C05405=1042.762,309.484,-115.253,172.109,41.467,157.953
C05406=1042.769,309.732,-115.287,172.114,41.469,157.954
C05407=1042.775,309.979,-115.320,172.118,41.472,157.955
C05408=1042.783,310.227,-115.354,172.122,41.474,157.956
C05409=1042.790,310.474,-115.386,172.126,41.477,157.956
C05410=1042.798,310.722,-115.420,172.129,41.479,157.957
C05411=1042.804,310.969,-115.454,172.133,41.482,157.958
C05412=1042.811,311.217,-115.487,172.137,41.484,157.959
C05413=1042.819,311.464,-115.521,172.141,41.487,157.960
C05414=1042.825,311.713,-115.554,172.145,41.489,157.960
C05415=1042.833,311.960,-115.588,172.149,41.492,157.961
C05416=1042.839,312.207,-115.622,172.153,41.494,157.962
C05417=1042.846,312.455,-115.656,172.158,41.497,157.963
C05418=1042.854,312.703,-115.689,172.162,41.499,157.964
C05419=1042.860,312.951,-115.724,172.166,41.503,157.965
C05420=1042.867,313.198,-115.757,172.170,41.505,157.965
C05421=1042.873,313.446,-115.792,172.174,41.508,157.966
C05422=1042.880,313.693,-115.825,172.178,41.510,157.967
C05423=1042.886,313.940,-115.860,172.181,41.513,157.968
C05424=1042.894,314.188,-115.894,172.186,41.516,157.969
C05425=1042.900,314.436,-115.928,172.190,41.519,157.970
C05426=1042.907,314.683,-115.962,172.193,41.521,157.970
C05427=1042.915,314.931,-115.996,172.197,41.524,157.971
C05428=1042.921,315.178,-116.031,172.202,41.527,157.972
C05429=1042.928,315.425,-116.065,172.205,41.530,157.973
C05430=1042.934,315.673,-116.099,172.210,41.532,157.974
C05431=1042.942,315.921,-116.133,172.214,41.535,157.975
C05432=1042.948,316.168,-116.168,172.218,41.538,157.976
C05433=1042.955,316.415,-116.202,172.222,41.540,157.976
C05434=1042.961,316.663,-116.236,172.226,41.543,157.977
C05435=1042.969,316.911,-116.270,172.230,41.546,157.978
C05436=1042.975,317.158,-116.305,172.234,41.549,157.979
C05437=1042.983,317.406,-116.339,172.238,41.551,157.980
C05438=1042.989,317.653,-116.374,172.243,41.554,157.981
C05439=1042.997,317.901,-116.408,172.247,41.557,157.982
C05440=1043.003,318.149,-116.442,172.251,41.560,157.982
C05441=1043.011,318.396,-116.477,172.255,41.563,157.983
C05442=1043.016,318.643,-116.511,172.259,41.565,157.984
C05443=1043.024,318.890,-116.545,172.263,41.568,157.985
C05444=1043.033,319.226,-116.592,172.270,41.572,157.986
C05445=1043.042,319.561,-116.639,172.275,41.576,157.988
C05446=1043.052,319.896,-116.685,172.280,41.579,157.989
C05447=1043.062,320.232,-116.733,172.287,41.583,157.990
C05448=1043.069,320.479,-116.766,172.291,41.586,157.991
C05449=1043.076,320.727,-116.802,172.295,41.589,157.992
C05450=1043.082,320.975,-116.836,172.299,41.592,157.993
C05451=1043.090,321.222,-116.871,172.304,41.595,157.994
C05452=1043.096,321.469,-116.906,172.308,41.597,157.994
C05453=1043.104,321.717,-116.939,172.312,41.600,157.995
C05454=1043.110,321.964,-116.975,172.316,41.603,157.996
C05455=1043.118,322.211,-117.009,172.321,41.606,157.997
C05456=1043.124,322.459,-117.044,172.325,41.608,157.998
C05457=1043.132,322.706,-117.078,172.329,41.612,157.999
C05458=1043.139,322.954,-117.114,172.333,41.614,158.000
C05459=1043.146,323.202,-117.147,172.338,41.617,158.001
C05460=1043.153,323.449,-117.183,172.342,41.620,158.002
C05461=1043.160,323.697,-117.218,172.346,41.623,158.003
C05462=1043.167,323.944,-117.252,172.350,41.626,158.003
C05463=1043.174,324.192,-117.287,172.355,41.629,158.004
C05464=1043.181,324.439,-117.321,172.359,41.631,158.005
C05465=1043.189,324.687,-117.357,172.364,41.634,158.006
C05466=1043.196,324.934,-117.391,172.369,41.637,158.007
C05467=1043.203,325.181,-117.426,172.373,41.640,158.008
C05468=1043.210,325.429,-117.462,172.377,41.643,158.009
C05469=1043.218,325.677,-117.496,172.382,41.645,158.010
C05470=1043.225,325.924,-117.532,172.386,41.649,158.011
C05471=1043.232,326.171,-117.566,172.390,41.652,158.012
C05472=1043.239,326.419,-117.601,172.395,41.654,158.013
C05473=1043.247,326.667,-117.635,172.399,41.657,158.014
C05474=1043.254,326.914,-117.671,172.403,41.660,158.014
C05475=1043.260,327.161,-117.706,172.408,41.663,158.015
C05476=1043.268,327.408,-117.740,172.412,41.666,158.016
C05477=1043.275,327.656,-117.776,172.416,41.669,158.017
C05478=1043.283,327.903,-117.811,172.422,41.672,158.018
C05479=1043.290,328.150,-117.846,172.425,41.675,158.019
C05480=1043.297,328.398,-117.882,172.431,41.678,158.020
C05481=1043.305,328.645,-117.916,172.435,41.681,158.021
C05482=1043.312,328.894,-117.952,172.439,41.683,158.022
C05483=1043.319,329.141,-117.987,172.444,41.686,158.023
C05484=1043.326,329.388,-118.022,172.448,41.689,158.024
C05485=1043.334,329.635,-118.058,172.452,41.693,158.025
C05486=1043.341,329.883,-118.093,172.457,41.696,158.026
C05487=1043.348,330.130,-118.128,172.461,41.699,158.027
C05488=1043.355,330.378,-118.164,172.467,41.702,158.028
C05489=1043.362,330.625,-118.199,172.471,41.705,158.029
C05490=1043.369,330.872,-118.234,172.475,41.708,158.030
C05491=1043.376,331.120,-118.271,172.480,41.711,158.031
C05492=1043.382,331.367,-118.306,172.484,41.714,158.032
C05493=1043.389,331.614,-118.342,172.489,41.717,158.033
C05494=1043.397,331.862,-118.378,172.493,41.720,158.034
C05495=1043.404,332.109,-118.413,172.498,41.723,158.035
C05496=1043.411,332.357,-118.449,172.503,41.726,158.036
C05497=1043.418,332.604,-118.485,172.507,41.730,158.037
C05498=1043.425,332.851,-118.520,172.512,41.733,158.038
C05499=1043.433,333.099,-118.556,172.516,41.736,158.039
C05500=1043.443,333.428,-118.604,172.523,41.740,158.040
C05501=1043.452,333.760,-118.651,172.528,41.744,158.041
C05502=1043.462,334.090,-118.699,172.535,41.749,158.043
C05503=1043.472,334.420,-118.747,172.541,41.753,158.044
C05504=1043.479,334.667,-118.783,172.546,41.756,158.045
C05505=1043.486,334.915,-118.818,172.551,41.759,158.046
C05506=1043.493,335.162,-118.854,172.555,41.762,158.047
C05507=1043.501,335.409,-118.890,172.560,41.765,158.048
C05508=1043.508,335.656,-118.926,172.564,41.768,158.049
C05509=1043.515,335.904,-118.962,172.569,41.772,158.050
C05510=1043.522,336.151,-118.998,172.574,41.775,158.051
C05511=1043.529,336.399,-119.034,172.578,41.778,158.052
C05512=1043.536,336.645,-119.070,172.583,41.782,158.053
C05513=1043.543,336.893,-119.107,172.588,41.785,158.054
C05514=1043.550,337.140,-119.143,172.593,41.788,158.055
C05515=1043.558,337.387,-119.179,172.598,41.792,158.057
C05516=1043.565,337.635,-119.216,172.602,41.795,158.058
C05517=1043.572,337.882,-119.252,172.608,41.798,158.059
C05518=1043.580,338.129,-119.288,172.612,41.801,158.060
C05519=1043.588,338.377,-119.324,172.617,41.804,158.061
C05520=1043.594,338.624,-119.361,172.621,41.808,158.062
C05521=1043.602,338.871,-119.397,172.626,41.811,158.063
C05522=1043.609,339.118,-119.433,172.631,41.815,158.064
C05523=1043.616,339.366,-119.469,172.636,41.818,158.065
C05524=1043.623,339.613,-119.506,172.640,41.821,158.066
C05525=1043.631,339.861,-119.542,172.645,41.824,158.067
C05526=1043.637,340.108,-119.578,172.651,41.828,158.068
C05527=1043.645,340.355,-119.615,172.655,41.831,158.069
C05528=1043.653,340.602,-119.651,172.660,41.835,158.070
C05529=1043.660,340.849,-119.687,172.665,41.838,158.072
C05530=1043.667,341.096,-119.724,172.670,41.841,158.073
C05531=1043.675,341.344,-119.760,172.675,41.845,158.074
C05532=1043.682,341.591,-119.797,172.679,41.848,158.075
C05533=1043.689,341.838,-119.834,172.685,41.851,158.076
C05534=1043.697,342.085,-119.870,172.689,41.855,158.077
C05535=1043.704,342.333,-119.907,172.694,41.858,158.078
C05536=1043.711,342.580,-119.944,172.699,41.862,158.079
C05537=1043.718,342.828,-119.980,172.704,41.865,158.080
C05538=1043.726,343.074,-120.017,172.709,41.869,158.081
C05539=1043.733,343.321,-120.054,172.714,41.872,158.082
C05540=1043.741,343.568,-120.091,172.719,41.875,158.084
C05541=1043.748,343.816,-120.128,172.724,41.879,158.085
C05542=1043.755,344.063,-120.165,172.729,41.883,158.086
C05543=1043.762,344.310,-120.201,172.734,41.886,158.087
C05544=1043.769,344.557,-120.239,172.739,41.889,158.088
C05545=1043.777,344.804,-120.275,172.744,41.893,158.089
C05546=1043.784,345.052,-120.312,172.749,41.896,158.090
C05547=1043.792,345.299,-120.348,172.754,41.900,158.092
C05548=1043.799,345.546,-120.386,172.759,41.904,158.093
C05549=1043.806,345.793,-120.424,172.764,41.907,158.094
C05550=1043.814,346.041,-120.460,172.769,41.911,158.095
C05551=1043.821,346.288,-120.497,172.775,41.914,158.096
C05552=1043.828,346.534,-120.534,172.779,41.918,158.097
C05553=1043.836,346.781,-120.571,172.784,41.921,158.099
C05554=1043.843,347.029,-120.608,172.790,41.925,158.100
C05555=1043.850,347.276,-120.646,172.795,41.929,158.101
C05556=1043.860,347.603,-120.695,172.802,41.933,158.102
C05557=1043.870,347.929,-120.744,172.809,41.938,158.104
C05558=1043.880,348.256,-120.793,172.815,41.943,158.106
C05559=1043.890,348.583,-120.842,172.821,41.947,158.107
C05560=1043.897,348.830,-120.880,172.827,41.952,158.108
C05561=1043.905,349.077,-120.917,172.832,41.955,158.109
C05562=1043.912,349.324,-120.954,172.838,41.959,158.111
C05563=1043.920,349.571,-120.992,172.843,41.962,158.112
C05564=1043.927,349.818,-121.029,172.847,41.966,158.113
C05565=1043.935,350.065,-121.066,172.853,41.969,158.114
C05566=1043.942,350.312,-121.104,172.858,41.973,158.115
C05567=1043.949,350.559,-121.141,172.864,41.977,158.117
C05568=1043.957,350.807,-121.179,172.869,41.980,158.118
C05569=1043.965,351.054,-121.217,172.874,41.985,158.119
C05570=1043.972,351.301,-121.255,172.879,41.988,158.120
C05571=1043.979,351.548,-121.292,172.884,41.992,158.121
C05572=1043.987,351.795,-121.329,172.890,41.996,158.123
C05573=1043.994,352.042,-121.367,172.895,41.999,158.124
C05574=1044.002,352.288,-121.405,172.901,42.003,158.125
C05575=1044.009,352.535,-121.443,172.905,42.007,158.126
C05576=1044.017,352.783,-121.481,172.911,42.011,158.128
C05577=1044.025,353.030,-121.519,172.916,42.015,158.129
C05578=1044.032,353.277,-121.556,172.922,42.019,158.130
C05579=1044.039,353.523,-121.595,172.927,42.022,158.131
C05580=1044.047,353.771,-121.632,172.933,42.026,158.133
C05581=1044.055,354.018,-121.670,172.938,42.030,158.134
C05582=1044.062,354.265,-121.708,172.944,42.034,158.135
C05583=1044.069,354.512,-121.746,172.948,42.038,158.136
C05584=1044.077,354.759,-121.784,172.954,42.042,158.138
C05585=1044.085,355.006,-121.822,172.959,42.046,158.139
C05586=1044.092,355.253,-121.860,172.965,42.049,158.140
C05587=1044.100,355.500,-121.898,172.970,42.053,158.142
C05588=1044.107,355.747,-121.936,172.976,42.057,158.143
C05589=1044.115,355.994,-121.975,172.981,42.061,158.144
C05590=1044.122,356.241,-122.012,172.987,42.065,158.145
C05591=1044.131,356.487,-122.050,172.992,42.069,158.147
C05592=1044.139,356.734,-122.088,172.998,42.073,158.148
C05593=1044.145,356.982,-122.126,173.003,42.077,158.149
C05594=1044.153,357.228,-122.165,173.009,42.081,158.151
C05595=1044.161,357.475,-122.203,173.015,42.085,158.152
C05596=1044.169,357.722,-122.242,173.020,42.089,158.153
C05597=1044.177,357.970,-122.279,173.026,42.093,158.155
C05598=1044.184,358.216,-122.318,173.031,42.096,158.156
C05599=1044.192,358.463,-122.356,173.037,42.100,158.157
C05600=1044.199,358.710,-122.395,173.042,42.105,158.158
C05601=1044.207,358.957,-122.433,173.048,42.109,158.160
C05602=1044.215,359.204,-122.472,173.054,42.113,158.161
C05603=1044.222,359.451,-122.510,173.059,42.117,158.162
C05604=1044.230,359.698,-122.549,173.065,42.121,158.164
C05605=1044.238,359.944,-122.587,173.070,42.125,158.165
C05606=1044.245,360.191,-122.626,173.076,42.129,158.166
C05607=1044.253,360.438,-122.665,173.082,42.133,158.168
C05608=1044.261,360.685,-122.703,173.087,42.138,158.169
C05609=1044.269,360.932,-122.741,173.093,42.142,158.171
C05610=1044.276,361.180,-122.781,173.099,42.146,158.172
C05611=1044.284,361.426,-122.820,173.104,42.150,158.173
C05612=1044.294,361.758,-122.871,173.112,42.155,158.175
C05613=1044.305,362.091,-122.923,173.120,42.161,158.177
C05614=1044.315,362.423,-122.976,173.128,42.166,158.179
C05615=1044.326,362.755,-123.028,173.135,42.172,158.181
C05616=1044.333,363.003,-123.068,173.141,42.177,158.182
C05617=1044.341,363.249,-123.106,173.147,42.181,158.184
C05618=1044.349,363.496,-123.146,173.153,42.185,158.185
C05619=1044.356,363.743,-123.184,173.159,42.189,158.186
C05620=1044.365,363.989,-123.223,173.165,42.193,158.188
C05621=1044.372,364.237,-123.262,173.170,42.198,158.189
C05622=1044.380,364.483,-123.301,173.176,42.202,158.191
C05623=1044.387,364.730,-123.341,173.182,42.206,158.192
C05624=1044.396,364.977,-123.380,173.187,42.211,158.193
C05625=1044.403,365.223,-123.420,173.194,42.215,158.195
C05626=1044.411,365.470,-123.458,173.200,42.219,158.196
C05627=1044.419,365.717,-123.498,173.206,42.224,158.198
C05628=1044.425,365.964,-123.537,173.212,42.228,158.199
C05629=1044.434,366.210,-123.576,173.217,42.232,158.201
C05630=1044.442,366.457,-123.616,173.223,42.237,158.202
C05631=1044.450,366.703,-123.655,173.230,42.241,158.204
C05632=1044.457,366.951,-123.694,173.235,42.245,158.205
C05633=1044.465,367.197,-123.734,173.241,42.250,158.207
C05634=1044.473,367.444,-123.774,173.247,42.255,158.208
C05635=1044.482,367.691,-123.813,173.254,42.258,158.209
C05636=1044.489,367.937,-123.852,173.260,42.263,158.211
C05637=1044.497,368.184,-123.892,173.265,42.268,158.212
C05638=1044.505,368.431,-123.931,173.271,42.272,158.214
C05639=1044.513,368.678,-123.970,173.278,42.277,158.215
C05640=1044.521,368.925,-124.010,173.284,42.281,158.217
C05641=1044.529,369.171,-124.050,173.289,42.285,158.218
C05642=1044.537,369.418,-124.089,173.296,42.290,158.220
C05643=1044.545,369.665,-124.129,173.302,42.294,158.221
C05644=1044.552,369.911,-124.168,173.308,42.299,158.223
C05645=1044.560,370.158,-124.208,173.314,42.303,158.224
C05646=1044.569,370.404,-124.248,173.321,42.308,158.226
C05647=1044.577,370.651,-124.288,173.327,42.312,158.227
C05648=1044.585,370.897,-124.328,173.333,42.317,158.229
C05649=1044.593,371.144,-124.367,173.339,42.321,158.230
C05650=1044.601,371.391,-124.407,173.345,42.327,158.232
C05651=1044.609,371.637,-124.448,173.352,42.331,158.234
C05652=1044.616,371.884,-124.488,173.358,42.336,158.235
C05653=1044.624,372.131,-124.528,173.364,42.340,158.237
C05654=1044.633,372.377,-124.568,173.371,42.345,158.238
C05655=1044.641,372.624,-124.608,173.377,42.350,158.240
C05656=1044.649,372.870,-124.648,173.383,42.354,158.241
C05657=1044.656,373.117,-124.688,173.389,42.359,158.243
C05658=1044.664,373.364,-124.729,173.395,42.364,158.245
C05659=1044.672,373.611,-124.769,173.402,42.368,158.246
C05660=1044.680,373.857,-124.810,173.408,42.373,158.248
C05661=1044.688,374.104,-124.849,173.414,42.378,158.249
C05662=1044.697,374.350,-124.889,173.421,42.383,158.251
C05663=1044.705,374.597,-124.930,173.427,42.388,158.253
C05664=1044.713,374.844,-124.970,173.434,42.393,158.254
C05665=1044.721,375.090,-125.011,173.440,42.397,158.256
C05666=1044.729,375.336,-125.052,173.447,42.402,158.258
C05667=1044.737,375.583,-125.092,173.453,42.407,158.259
C05668=1044.748,375.935,-125.150,173.462,42.414,158.261
C05669=1044.760,376.287,-125.207,173.472,42.421,158.264
C05670=1044.772,376.639,-125.266,173.481,42.427,158.266
C05671=1044.783,376.991,-125.324,173.490,42.434,158.268
C05672=1044.792,377.237,-125.364,173.497,42.439,158.270
C05673=1044.800,377.483,-125.404,173.504,42.444,158.272
C05674=1044.809,377.730,-125.445,173.510,42.449,158.273
C05675=1044.817,377.976,-125.486,173.517,42.454,158.275
C05676=1044.825,378.223,-125.527,173.524,42.459,158.277
C05677=1044.833,378.470,-125.568,173.530,42.464,158.278
C05678=1044.841,378.716,-125.608,173.537,42.469,158.280
C05679=1044.849,378.962,-125.649,173.543,42.474,158.282
C05680=1044.858,379.209,-125.690,173.550,42.479,158.283
C05681=1044.866,379.455,-125.730,173.557,42.484,158.285
C05682=1044.874,379.702,-125.771,173.563,42.489,158.287
C05683=1044.882,379.948,-125.813,173.570,42.494,158.289
C05684=1044.890,380.195,-125.854,173.576,42.499,158.290
C05685=1044.898,380.441,-125.895,173.584,42.504,158.292
C05686=1044.907,380.687,-125.936,173.591,42.509,158.294
C05687=1044.915,380.934,-125.978,173.597,42.514,158.296
C05688=1044.924,381.180,-126.019,173.604,42.519,158.297
C05689=1044.932,381.427,-126.060,173.610,42.525,158.299
C05690=1044.940,381.674,-126.101,173.617,42.530,158.301
C05691=1044.948,381.920,-126.143,173.624,42.535,158.303
C05692=1044.956,382.165,-126.184,173.632,42.540,158.304
C05693=1044.965,382.412,-126.225,173.638,42.545,158.306
C05694=1044.973,382.658,-126.267,173.645,42.550,158.308
C05695=1044.981,382.905,-126.308,173.652,42.556,158.310
C05696=1044.990,383.151,-126.350,173.658,42.561,158.311
C05697=1044.998,383.397,-126.391,173.666,42.566,158.313
C05698=1045.006,383.644,-126.433,173.673,42.571,158.315
C05699=1045.014,383.890,-126.474,173.680,42.577,158.317
C05700=1045.023,384.136,-126.516,173.686,42.582,158.319
C05701=1045.032,384.382,-126.557,173.694,42.587,158.320
C05702=1045.040,384.629,-126.599,173.701,42.593,158.322
C05703=1045.049,384.876,-126.641,173.708,42.598,158.324
C05704=1045.057,385.121,-126.682,173.714,42.603,158.326
C05705=1045.065,385.368,-126.724,173.722,42.609,158.328
C05706=1045.074,385.615,-126.766,173.729,42.614,158.330
C05707=1045.082,385.860,-126.807,173.736,42.620,158.332
C05708=1045.091,386.107,-126.849,173.743,42.625,158.333
C05709=1045.099,386.353,-126.891,173.751,42.630,158.335
C05710=1045.108,386.600,-126.933,173.757,42.636,158.337
C05711=1045.117,386.845,-126.974,173.764,42.641,158.339
C05712=1045.125,387.092,-127.017,173.772,42.647,158.341
C05713=1045.134,387.338,-127.058,173.779,42.652,158.343
C05714=1045.143,387.585,-127.100,173.786,42.658,158.345
C05715=1045.151,387.831,-127.143,173.794,42.663,158.347
C05716=1045.160,388.077,-127.185,173.801,42.669,158.348
C05717=1045.169,388.323,-127.226,173.808,42.674,158.350
C05718=1045.177,388.569,-127.269,173.816,42.679,158.352
C05719=1045.186,388.815,-127.311,173.823,42.685,158.354
C05720=1045.194,389.062,-127.353,173.831,42.691,158.356
C05721=1045.203,389.308,-127.395,173.838,42.696,158.358
C05722=1045.212,389.554,-127.438,173.844,42.702,158.360
C05723=1045.220,389.801,-127.480,173.852,42.708,158.362
C05724=1045.231,390.093,-127.531,173.861,42.714,158.364
C05725=1045.241,390.386,-127.581,173.870,42.721,158.367
C05726=1045.251,390.679,-127.632,173.879,42.728,158.369
C05727=1045.261,390.971,-127.682,173.888,42.735,158.371
C05728=1045.270,391.218,-127.725,173.895,42.740,158.373
C05729=1045.279,391.464,-127.767,173.903,42.746,158.375
C05730=1045.287,391.710,-127.810,173.910,42.752,158.377
C05731=1045.296,391.956,-127.853,173.917,42.758,158.379
C05732=1045.305,392.202,-127.895,173.925,42.763,158.381
C05733=1045.313,392.448,-127.938,173.934,42.769,158.383
C05734=1045.322,392.694,-127.981,173.941,42.775,158.385
C05735=1045.331,392.941,-128.024,173.949,42.781,158.387
C05736=1045.340,393.187,-128.067,173.956,42.787,158.389
C05737=1045.349,393.433,-128.110,173.964,42.793,158.391
C05738=1045.357,393.679,-128.153,173.971,42.799,158.394
C05739=1045.366,393.925,-128.196,173.979,42.805,158.396
C05740=1045.375,394.171,-128.238,173.987,42.811,158.398
C05741=1045.383,394.417,-128.281,173.994,42.817,158.400
C05742=1045.392,394.663,-128.325,174.003,42.822,158.402
C05743=1045.401,394.910,-128.368,174.010,42.828,158.404
C05744=1045.411,395.155,-128.411,174.018,42.834,158.406
C05745=1045.419,395.401,-128.454,174.026,42.840,158.408
C05746=1045.428,395.647,-128.497,174.033,42.846,158.410
C05747=1045.437,395.893,-128.540,174.042,42.852,158.412
C05748=1045.445,396.139,-128.584,174.050,42.858,158.414
C05749=1045.454,396.385,-128.627,174.057,42.864,158.417
C05750=1045.463,396.631,-128.671,174.065,42.871,158.419
C05751=1045.472,396.877,-128.714,174.074,42.877,158.421
C05752=1045.481,397.123,-128.758,174.081,42.883,158.423
C05753=1045.490,397.369,-128.801,174.089,42.889,158.425
C05754=1045.499,397.615,-128.845,174.097,42.895,158.427
C05755=1045.508,397.862,-128.889,174.106,42.901,158.430
C05756=1045.516,398.107,-128.932,174.114,42.908,158.432
C05757=1045.526,398.352,-128.975,174.121,42.914,158.434
C05758=1045.535,398.599,-129.019,174.130,42.920,158.436
C05759=1045.544,398.844,-129.063,174.138,42.926,158.438
C05760=1045.553,399.090,-129.107,174.145,42.932,158.440
C05761=1045.562,399.336,-129.150,174.154,42.939,158.443
C05762=1045.571,399.583,-129.194,174.162,42.945,158.445
C05763=1045.580,399.828,-129.238,174.171,42.952,158.447
C05764=1045.589,400.074,-129.282,174.179,42.957,158.449
C05765=1045.599,400.320,-129.326,174.187,42.964,158.452
C05766=1045.608,400.566,-129.370,174.195,42.970,158.454
C05767=1045.616,400.812,-129.414,174.203,42.977,158.456
C05768=1045.625,401.058,-129.458,174.212,42.983,158.458
C05769=1045.635,401.304,-129.502,174.220,42.989,158.461
C05770=1045.644,401.550,-129.546,174.229,42.996,158.463
C05771=1045.653,401.795,-129.590,174.237,43.003,158.465
C05772=1045.662,402.041,-129.634,174.246,43.009,158.468
C05773=1045.671,402.287,-129.679,174.254,43.015,158.470
C05774=1045.681,402.533,-129.724,174.263,43.022,158.472
C05775=1045.689,402.779,-129.767,174.271,43.029,158.475
C05776=1045.702,403.117,-129.829,174.283,43.037,158.478
C05777=1045.715,403.456,-129.890,174.294,43.047,158.481
C05778=1045.728,403.793,-129.951,174.306,43.056,158.484
C05779=1045.740,404.131,-130.012,174.318,43.065,158.488
C05780=1045.756,404.536,-130.086,174.332,43.076,158.492
C05781=1045.770,404.941,-130.160,174.346,43.087,158.496
C05782=1045.786,405.345,-130.233,174.360,43.098,158.500
C05783=1045.802,405.749,-130.307,174.376,43.109,158.504
C05784=1045.810,405.995,-130.353,174.384,43.116,158.506
C05785=1045.820,406.241,-130.397,174.393,43.123,158.508
C05786=1045.829,406.487,-130.442,174.402,43.130,158.511
C05787=1045.839,406.732,-130.487,174.410,43.137,158.513
C05788=1045.848,406.978,-130.532,174.419,43.144,158.516
C05789=1045.857,407.223,-130.577,174.428,43.150,158.518
C05790=1045.866,407.469,-130.623,174.438,43.157,158.521
C05791=1045.876,407.715,-130.667,174.447,43.164,158.523
C05792=1045.885,407.961,-130.713,174.455,43.172,158.526
C05793=1045.895,408.206,-130.758,174.464,43.178,158.528
C05794=1045.904,408.452,-130.802,174.473,43.185,158.531
C05795=1045.914,408.697,-130.849,174.483,43.192,158.533
C05796=1045.924,408.943,-130.894,174.492,43.199,158.536
C05797=1045.933,409.189,-130.939,174.500,43.207,158.539
C05798=1045.943,409.434,-130.984,174.509,43.213,158.541
C05799=1045.952,409.680,-131.030,174.519,43.221,158.544
C05800=1045.962,409.926,-131.075,174.528,43.228,158.546
C05801=1045.971,410.172,-131.121,174.537,43.235,158.549
C05802=1045.981,410.417,-131.166,174.547,43.242,158.552
C05803=1045.991,410.663,-131.212,174.556,43.249,158.554
C05804=1046.001,410.908,-131.258,174.565,43.256,158.557
C05805=1046.010,411.155,-131.303,174.575,43.263,158.559
C05806=1046.020,411.400,-131.350,174.584,43.271,158.562
C05807=1046.030,411.645,-131.395,174.594,43.278,158.565
C05808=1046.039,411.891,-131.441,174.603,43.285,158.567
C05809=1046.050,412.137,-131.487,174.613,43.292,158.570
C05810=1046.059,412.383,-131.532,174.622,43.300,158.573
C05811=1046.070,412.628,-131.578,174.631,43.307,158.575
C05812=1046.079,412.873,-131.624,174.641,43.315,158.578
C05813=1046.089,413.119,-131.671,174.650,43.322,158.581
C05814=1046.098,413.364,-131.717,174.661,43.329,158.583
C05815=1046.108,413.610,-131.763,174.671,43.337,158.586
C05816=1046.117,413.856,-131.810,174.680,43.344,158.589
C05817=1046.128,414.101,-131.855,174.690,43.352,158.592
C05818=1046.137,414.346,-131.902,174.699,43.359,158.594
C05819=1046.147,414.592,-131.948,174.709,43.367,158.597
C05820=1046.157,414.838,-131.995,174.719,43.375,158.600
C05821=1046.166,415.083,-132.041,174.729,43.382,158.603
C05822=1046.176,415.329,-132.088,174.739,43.389,158.606
C05823=1046.186,415.575,-132.134,174.748,43.397,158.608
C05824=1046.197,415.819,-132.181,174.758,43.405,158.611
C05825=1046.206,416.065,-132.227,174.769,43.412,158.614
C05826=1046.217,416.310,-132.274,174.778,43.420,158.617
C05827=1046.227,416.556,-132.321,174.788,43.428,158.620
C05828=1046.236,416.801,-132.368,174.799,43.436,158.623
C05829=1046.246,417.046,-132.414,174.809,43.443,158.626
C05830=1046.256,417.292,-132.461,174.818,43.451,158.628
C05831=1046.266,417.538,-132.508,174.829,43.459,158.631
C05832=1046.277,417.783,-132.555,174.839,43.466,158.634
C05833=1046.287,418.028,-132.602,174.850,43.474,158.637
C05834=1046.297,418.274,-132.648,174.859,43.482,158.640
C05835=1046.307,418.519,-132.695,174.870,43.490,158.643
C05836=1046.324,418.930,-132.775,174.888,43.503,158.648
C05837=1046.341,419.343,-132.855,174.904,43.517,158.653
C05838=1046.358,419.754,-132.934,174.922,43.530,158.658
C05839=1046.375,420.166,-133.014,174.940,43.544,158.663
C05840=1046.386,420.412,-133.061,174.951,43.552,158.666
C05841=1046.396,420.657,-133.108,174.962,43.560,158.669
C05842=1046.405,420.902,-133.156,174.972,43.568,158.672
C05843=1046.416,421.147,-133.204,174.983,43.576,158.676
C05844=1046.426,421.392,-133.251,174.994,43.584,158.679
C05845=1046.436,421.638,-133.298,175.004,43.593,158.682
C05846=1046.447,421.883,-133.347,175.015,43.601,158.685
C05847=1046.457,422.128,-133.394,175.026,43.609,158.688
C05848=1046.467,422.373,-133.442,175.036,43.617,158.691
C05849=1046.477,422.619,-133.490,175.047,43.625,158.694
C05850=1046.489,422.864,-133.538,175.058,43.634,158.697
C05851=1046.499,423.109,-133.586,175.069,43.642,158.700
C05852=1046.509,423.354,-133.633,175.080,43.651,158.704
C05853=1046.520,423.599,-133.681,175.090,43.659,158.707
C05854=1046.530,423.844,-133.730,175.102,43.667,158.710
C05855=1046.541,424.090,-133.778,175.113,43.676,158.713
C05856=1046.552,424.334,-133.826,175.124,43.684,158.717
C05857=1046.562,424.580,-133.874,175.135,43.693,158.720
C05858=1046.572,424.825,-133.922,175.147,43.701,158.723
C05859=1046.583,425.071,-133.970,175.158,43.710,158.726
C05860=1046.594,425.315,-134.019,175.169,43.718,158.730
C05861=1046.604,425.560,-134.068,175.181,43.727,158.733
C05862=1046.615,425.805,-134.116,175.192,43.735,158.736
C05863=1046.625,426.051,-134.165,175.203,43.744,158.739
C05864=1046.636,426.296,-134.213,175.215,43.753,158.743
C05865=1046.647,426.540,-134.262,175.226,43.761,158.746
C05866=1046.658,426.786,-134.311,175.238,43.770,158.750
C05867=1046.668,427.030,-134.359,175.249,43.779,158.753
C05868=1046.679,427.275,-134.408,175.261,43.788,158.756
C05869=1046.690,427.520,-134.457,175.273,43.797,158.760
C05870=1046.701,427.766,-134.506,175.284,43.805,158.763
C05871=1046.711,428.010,-134.555,175.296,43.814,158.767
C05872=1046.723,428.255,-134.604,175.308,43.823,158.770
C05873=1046.733,428.500,-134.653,175.319,43.832,158.773
C05874=1046.744,428.745,-134.702,175.332,43.841,158.777
C05875=1046.755,428.990,-134.751,175.343,43.850,158.780
C05876=1046.766,429.235,-134.801,175.355,43.859,158.784
C05877=1046.777,429.479,-134.850,175.368,43.868,158.787
C05878=1046.787,429.724,-134.899,175.379,43.877,158.791
C05879=1046.798,429.969,-134.949,175.391,43.886,158.794
C05880=1046.809,430.214,-134.998,175.404,43.895,158.798
C05881=1046.820,430.459,-135.047,175.416,43.904,158.802
C05882=1046.831,430.704,-135.097,175.427,43.914,158.805
C05883=1046.842,430.948,-135.147,175.440,43.922,158.809
C05884=1046.853,431.193,-135.196,175.452,43.932,158.812
C05885=1046.864,431.438,-135.246,175.465,43.941,158.816
C05886=1046.875,431.683,-135.296,175.477,43.951,158.820
C05887=1046.886,431.928,-135.345,175.490,43.960,158.823
C05888=1046.897,432.172,-135.396,175.502,43.969,158.827
C05889=1046.908,432.418,-135.446,175.514,43.979,158.831
C05890=1046.920,432.662,-135.495,175.527,43.988,158.835
C05891=1046.931,432.907,-135.545,175.539,43.997,158.838
C05892=1046.941,433.124,-135.590,175.551,44.006,158.841
C05893=1046.951,433.342,-135.634,175.562,44.014,158.845
C05894=1046.961,433.559,-135.679,175.573,44.022,158.848
C05895=1046.971,433.776,-135.724,175.585,44.030,158.851
C05896=1046.981,433.993,-135.767,175.596,44.039,158.855
C05897=1046.991,434.210,-135.812,175.608,44.048,158.858
C05898=1047.001,434.428,-135.857,175.618,44.056,158.862
C05899=1047.012,434.644,-135.902,175.630,44.065,158.865
C05900=1047.023,434.889,-135.952,175.643,44.074,158.869
C05901=1047.034,435.134,-136.003,175.656,44.084,158.873
C05902=1047.045,435.378,-136.053,175.669,44.094,158.877
C05903=1047.058,435.623,-136.103,175.683,44.103,158.880
C05904=1047.069,435.868,-136.154,175.696,44.113,158.884
C05905=1047.080,436.112,-136.205,175.709,44.123,158.888
C05906=1047.092,436.357,-136.256,175.722,44.133,158.892
C05907=1047.103,436.601,-136.307,175.736,44.142,158.896
C05908=1047.115,436.846,-136.357,175.749,44.152,158.900
C05909=1047.126,437.090,-136.408,175.762,44.162,158.904
C05910=1047.138,437.335,-136.459,175.776,44.172,158.908
C05911=1047.150,437.580,-136.511,175.789,44.182,158.912
C05912=1047.161,437.824,-136.562,175.803,44.192,158.916
C05913=1047.173,438.068,-136.613,175.817,44.202,158.920
C05914=1047.184,438.313,-136.664,175.831,44.212,158.925
C05915=1047.196,438.558,-136.715,175.844,44.223,158.929
C05916=1047.208,438.802,-136.766,175.858,44.233,158.933
C05917=1047.219,439.046,-136.818,175.872,44.243,158.937
C05918=1047.232,439.290,-136.870,175.886,44.253,158.941
C05919=1047.243,439.534,-136.921,175.900,44.263,158.945
C05920=1047.255,439.779,-136.972,175.914,44.273,158.949
C05921=1047.267,440.023,-137.024,175.928,44.283,158.954
C05922=1047.279,440.268,-137.075,175.941,44.294,158.958
C05923=1047.291,440.512,-137.127,175.956,44.304,158.962
C05924=1047.303,440.756,-137.179,175.970,44.314,158.966
C05925=1047.315,441.000,-137.231,175.985,44.325,158.971
C05926=1047.327,441.245,-137.282,175.998,44.335,158.975
C05927=1047.339,441.490,-137.335,176.013,44.346,158.979
C05928=1047.351,441.733,-137.388,176.028,44.356,158.984
C05929=1047.363,441.978,-137.439,176.042,44.367,158.988
C05930=1047.376,442.222,-137.491,176.057,44.378,158.992
C05931=1047.388,442.466,-137.543,176.071,44.388,158.997
C05932=1047.399,442.710,-137.596,176.086,44.399,159.001
C05933=1047.412,442.955,-137.648,176.101,44.409,159.006
C05934=1047.424,443.198,-137.700,176.116,44.420,159.010
C05935=1047.436,443.442,-137.753,176.130,44.431,159.014
C05936=1047.448,443.687,-137.806,176.145,44.442,159.019
C05937=1047.461,443.931,-137.858,176.160,44.452,159.023
C05938=1047.473,444.174,-137.911,176.175,44.463,159.028
C05939=1047.486,444.419,-137.963,176.191,44.474,159.033
C05940=1047.497,444.663,-138.016,176.206,44.485,159.037
C05941=1047.510,444.907,-138.069,176.221,44.496,159.042
C05942=1047.523,445.151,-138.121,176.236,44.507,159.046
C05943=1047.536,445.395,-138.174,176.252,44.518,159.051
C05944=1047.548,445.638,-138.227,176.267,44.529,159.056
C05945=1047.561,445.880,-138.279,176.282,44.540,159.060
C05946=1047.575,446.124,-138.332,176.298,44.550,159.065
C05947=1047.589,446.368,-138.383,176.314,44.561,159.069
C05948=1047.604,446.612,-138.434,176.330,44.571,159.074
C05949=1047.620,446.855,-138.484,176.345,44.582,159.078
C05950=1047.636,447.099,-138.534,176.361,44.592,159.083
C05951=1047.654,447.343,-138.583,176.377,44.602,159.087
C05952=1047.680,447.713,-138.657,176.401,44.617,159.094
C05953=1047.709,448.082,-138.729,176.425,44.632,159.101
C05954=1047.739,448.452,-138.800,176.450,44.646,159.107
C05955=1047.771,448.823,-138.871,176.474,44.660,159.114
C05956=1047.793,449.067,-138.917,176.491,44.669,159.118
C05957=1047.815,449.312,-138.962,176.508,44.678,159.122
C05958=1047.838,449.558,-139.006,176.525,44.687,159.126
C05959=1047.862,449.802,-139.051,176.541,44.696,159.131
C05960=1047.886,450.048,-139.094,176.558,44.704,159.135
C05961=1047.911,450.294,-139.138,176.575,44.713,159.139
C05962=1047.937,450.539,-139.180,176.592,44.721,159.143
C05963=1047.964,450.783,-139.222,176.609,44.729,159.147
C05964=1047.654,450.817,-139.527,176.610,44.817,159.173
C05965=1047.628,450.571,-139.485,176.593,44.809,159.169
C05966=1047.602,450.325,-139.443,176.575,44.801,159.165
C05967=1047.576,450.080,-139.399,176.559,44.792,159.161
C05968=1047.552,449.835,-139.356,176.542,44.784,159.157
C05969=1047.528,449.590,-139.312,176.525,44.775,159.152
C05970=1047.505,449.344,-139.267,176.508,44.767,159.148
C05971=1047.482,449.100,-139.222,176.492,44.757,159.144
C05972=1047.460,448.854,-139.176,176.475,44.748,159.140
C05973=1047.430,448.502,-139.110,176.451,44.735,159.133
C05974=1047.401,448.149,-139.042,176.428,44.722,159.127
C05975=1047.373,447.797,-138.973,176.404,44.708,159.121
C05976=1047.346,447.445,-138.904,176.381,44.694,159.114
C05977=1047.330,447.201,-138.854,176.365,44.684,159.110
C05978=1047.312,446.957,-138.804,176.349,44.674,159.105
C05979=1047.296,446.713,-138.754,176.333,44.664,159.101
C05980=1047.280,446.469,-138.704,176.317,44.654,159.096
C05981=1047.266,446.226,-138.653,176.302,44.643,159.092
C05982=1047.252,445.982,-138.601,176.287,44.632,159.087
C05983=1047.239,445.739,-138.549,176.270,44.622,159.083
C05984=1047.225,445.496,-138.497,176.255,44.611,159.078
C05985=1047.213,445.252,-138.444,176.240,44.600,159.073
C05986=1047.201,445.008,-138.390,176.224,44.589,159.069
C05987=1047.188,444.764,-138.338,176.209,44.578,159.064
C05988=1047.175,444.520,-138.285,176.194,44.567,159.060
C05989=1047.163,444.276,-138.233,176.179,44.557,159.055
C05990=1047.150,444.032,-138.180,176.164,44.546,159.051
C05991=1047.139,443.788,-138.127,176.148,44.535,159.046
C05992=1047.126,443.544,-138.074,176.133,44.524,159.041
C05993=1047.114,443.300,-138.022,176.118,44.514,159.037
C05994=1047.101,443.056,-137.970,176.103,44.503,159.033
C05995=1047.089,442.811,-137.917,176.089,44.493,159.028
C05996=1047.077,442.567,-137.865,176.074,44.482,159.024
C05997=1047.065,442.323,-137.813,176.059,44.471,159.019
C05998=1047.053,442.079,-137.761,176.044,44.461,159.015
C05999=1047.041,441.835,-137.709,176.030,44.450,159.010
C06000=1047.028,441.590,-137.655,176.015,44.440,159.006
C06001=1047.017,441.346,-137.604,176.000,44.429,159.002
C06002=1047.004,441.102,-137.552,175.986,44.419,158.997
C06003=1046.993,440.858,-137.501,175.972,44.409,158.993
C06004=1046.980,440.614,-137.448,175.958,44.398,158.989
C06005=1046.968,440.369,-137.397,175.943,44.388,158.985
C06006=1046.956,440.125,-137.345,175.929,44.378,158.980
C06007=1046.944,439.881,-137.293,175.915,44.368,158.976
C06008=1046.933,439.636,-137.242,175.901,44.357,158.972
C06009=1046.920,439.392,-137.190,175.887,44.347,158.968
C06010=1046.908,439.148,-137.139,175.873,44.337,158.964
C06011=1046.897,438.903,-137.087,175.859,44.327,158.959
C06012=1046.885,438.659,-137.035,175.845,44.317,158.955
C06013=1046.874,438.414,-136.984,175.831,44.307,158.951
C06014=1046.862,438.170,-136.933,175.818,44.297,158.947
C06015=1046.850,437.926,-136.881,175.804,44.287,158.943
C06016=1046.839,437.681,-136.831,175.790,44.277,158.939
C06017=1046.826,437.436,-136.780,175.776,44.267,158.935
C06018=1046.815,437.193,-136.729,175.763,44.257,158.931
C06019=1046.803,436.948,-136.677,175.749,44.247,158.927
C06020=1046.791,436.703,-136.627,175.736,44.238,158.923
C06021=1046.780,436.459,-136.576,175.723,44.228,158.919
C06022=1046.769,436.214,-136.525,175.709,44.218,158.915
C06023=1046.757,435.970,-136.474,175.696,44.208,158.911
C06024=1046.746,435.725,-136.423,175.683,44.198,158.907
C06025=1046.734,435.480,-136.372,175.669,44.189,158.903
C06026=1046.722,435.236,-136.323,175.656,44.180,158.899
C06027=1046.711,434.991,-136.271,175.643,44.170,158.895
C06028=1046.700,434.747,-136.221,175.630,44.160,158.892
C06029=1046.689,434.528,-136.176,175.618,44.152,158.888
C06030=1046.679,434.311,-136.131,175.607,44.143,158.885
C06031=1046.669,434.092,-136.086,175.595,44.135,158.881
C06032=1046.658,433.874,-136.042,175.584,44.127,158.878
C06033=1046.649,433.656,-135.997,175.572,44.118,158.875
C06034=1046.638,433.438,-135.952,175.560,44.109,158.871
C06035=1046.628,433.219,-135.907,175.549,44.101,158.868
C06036=1046.618,433.001,-135.863,175.539,44.093,158.865
C06037=1046.607,432.757,-135.812,175.526,44.083,158.861
C06038=1046.595,432.512,-135.763,175.513,44.074,158.857
C06039=1046.585,432.267,-135.713,175.501,44.065,158.853
C06040=1046.574,432.022,-135.663,175.488,44.055,158.850
C06041=1046.562,431.777,-135.613,175.475,44.046,158.846
C06042=1046.551,431.532,-135.564,175.463,44.037,158.842
C06043=1046.540,431.288,-135.513,175.450,44.028,158.839
C06044=1046.529,431.043,-135.464,175.438,44.019,158.835
C06045=1046.518,430.798,-135.415,175.425,44.009,158.831
C06046=1046.507,430.554,-135.364,175.414,44.000,158.828
C06047=1046.496,430.309,-135.315,175.401,43.991,158.824
C06048=1046.485,430.064,-135.266,175.389,43.982,158.821
C06049=1046.474,429.819,-135.216,175.376,43.973,158.817
C06050=1046.463,429.574,-135.167,175.365,43.964,158.814
C06051=1046.452,429.329,-135.118,175.353,43.955,158.810
C06052=1046.442,429.085,-135.068,175.340,43.946,158.807
C06053=1046.431,428.840,-135.019,175.329,43.937,158.803
C06054=1046.420,428.595,-134.970,175.317,43.928,158.800
C06055=1046.409,428.350,-134.920,175.304,43.920,158.796
C06056=1046.398,428.105,-134.872,175.293,43.911,158.793
C06057=1046.387,427.860,-134.822,175.281,43.902,158.789
C06058=1046.376,427.615,-134.773,175.270,43.893,158.786
C06059=1046.366,427.370,-134.725,175.257,43.885,158.782
C06060=1046.355,427.125,-134.676,175.246,43.876,158.779
C06061=1046.344,426.880,-134.627,175.234,43.867,158.776
C06062=1046.333,426.635,-134.578,175.223,43.859,158.772
C06063=1046.323,426.390,-134.530,175.211,43.850,158.769
C06064=1046.312,426.144,-134.481,175.200,43.841,158.766
C06065=1046.301,425.900,-134.432,175.189,43.833,158.762
C06066=1046.290,425.655,-134.384,175.177,43.824,158.759
C06067=1046.280,425.409,-134.335,175.166,43.815,158.755
C06068=1046.270,425.165,-134.287,175.154,43.807,158.752
C06069=1046.259,424.920,-134.238,175.143,43.798,158.749
C06070=1046.248,424.675,-134.190,175.132,43.790,158.746
C06071=1046.238,424.429,-134.142,175.120,43.781,158.742
C06072=1046.227,424.184,-134.094,175.109,43.773,158.739
C06073=1046.216,423.939,-134.046,175.098,43.765,158.736
C06074=1046.206,423.694,-133.997,175.087,43.756,158.733
C06075=1046.195,423.449,-133.949,175.076,43.748,158.730
C06076=1046.185,423.204,-133.901,175.064,43.740,158.726
C06077=1046.174,422.959,-133.854,175.053,43.732,158.723
C06078=1046.163,422.713,-133.806,175.042,43.723,158.720
C06079=1046.154,422.468,-133.757,175.032,43.715,158.717
C06080=1046.143,422.223,-133.710,175.021,43.707,158.714
C06081=1046.132,421.978,-133.661,175.010,43.698,158.711
C06082=1046.122,421.732,-133.614,174.999,43.690,158.707
C06083=1046.112,421.488,-133.566,174.988,43.682,158.704
C06084=1046.101,421.242,-133.519,174.977,43.674,158.701
C06085=1046.091,420.996,-133.471,174.966,43.666,158.698
C06086=1046.081,420.751,-133.423,174.956,43.658,158.695
C06087=1046.071,420.506,-133.376,174.945,43.650,158.692
C06088=1046.060,420.261,-133.329,174.934,43.642,158.689
C06089=1046.044,419.847,-133.248,174.917,43.628,158.684
C06090=1046.026,419.434,-133.169,174.899,43.615,158.679
C06091=1046.009,419.020,-133.088,174.881,43.602,158.674
C06092=1045.992,418.606,-133.009,174.864,43.588,158.669
C06093=1045.982,418.361,-132.962,174.854,43.580,158.666
C06094=1045.972,418.115,-132.915,174.843,43.573,158.663
C06095=1045.962,417.870,-132.868,174.833,43.565,158.660
C06096=1045.952,417.624,-132.821,174.823,43.557,158.657
C06097=1045.941,417.379,-132.774,174.813,43.549,158.654
C06098=1045.931,417.134,-132.727,174.802,43.541,158.651
C06099=1045.921,416.888,-132.681,174.792,43.534,158.648
C06100=1045.910,416.643,-132.634,174.782,43.526,158.645
C06101=1045.901,416.397,-132.587,174.772,43.518,158.643
C06102=1045.891,416.152,-132.540,174.762,43.511,158.640
C06103=1045.881,415.906,-132.494,174.752,43.504,158.637
C06104=1045.871,415.660,-132.447,174.742,43.496,158.634
C06105=1045.861,415.415,-132.400,174.732,43.488,158.631
C06106=1045.851,415.170,-132.354,174.722,43.480,158.628
C06107=1045.841,414.924,-132.308,174.712,43.473,158.626
C06108=1045.831,414.679,-132.261,174.702,43.466,158.623
C06109=1045.822,414.434,-132.215,174.692,43.458,158.620
C06110=1045.812,414.188,-132.168,174.683,43.451,158.617
C06111=1045.802,413.942,-132.122,174.673,43.443,158.614
C06112=1045.792,413.697,-132.076,174.663,43.436,158.612
C06113=1045.782,413.451,-132.030,174.653,43.429,158.609
C06114=1045.773,413.206,-131.983,174.643,43.421,158.606
C06115=1045.763,412.960,-131.937,174.634,43.414,158.604
C06116=1045.753,412.715,-131.891,174.625,43.406,158.601
C06117=1045.744,412.469,-131.844,174.615,43.399,158.598
C06118=1045.734,412.224,-131.799,174.606,43.392,158.595
C06119=1045.724,411.978,-131.752,174.596,43.385,158.593
C06120=1045.713,411.732,-131.707,174.587,43.377,158.590
C06121=1045.704,411.487,-131.661,174.576,43.370,158.587
C06122=1045.694,411.241,-131.616,174.567,43.363,158.585
C06123=1045.685,410.995,-131.570,174.557,43.356,158.582
C06124=1045.674,410.750,-131.524,174.548,43.348,158.579
C06125=1045.665,410.504,-131.478,174.539,43.342,158.577
C06126=1045.655,410.259,-131.433,174.529,43.334,158.574
C06127=1045.646,410.013,-131.387,174.520,43.327,158.572
C06128=1045.636,409.767,-131.342,174.511,43.320,158.569
C06129=1045.626,409.522,-131.296,174.502,43.313,158.566
C06130=1045.617,409.276,-131.251,174.493,43.306,158.564
C06131=1045.607,409.030,-131.205,174.484,43.299,158.561
C06132=1045.597,408.785,-131.160,174.474,43.292,158.559
C06133=1045.588,408.539,-131.114,174.465,43.285,158.556
C06134=1045.578,408.293,-131.070,174.456,43.278,158.554
C06135=1045.569,408.048,-131.024,174.447,43.271,158.551
C06136=1045.559,407.801,-130.979,174.437,43.265,158.549
C06137=1045.550,407.556,-130.934,174.429,43.258,158.546
C06138=1045.540,407.310,-130.889,174.420,43.250,158.544
C06139=1045.531,407.064,-130.843,174.411,43.244,158.541
C06140=1045.522,406.819,-130.798,174.401,43.237,158.539
C06141=1045.512,406.573,-130.754,174.393,43.230,158.536
C06142=1045.503,406.327,-130.708,174.384,43.223,158.534
C06143=1045.493,406.082,-130.663,174.375,43.216,158.531
C06144=1045.484,405.836,-130.618,174.366,43.210,158.529
C06145=1045.469,405.430,-130.544,174.352,43.199,158.525
C06146=1045.454,405.023,-130.470,174.338,43.188,158.521
C06147=1045.438,404.617,-130.396,174.322,43.176,158.517
C06148=1045.423,404.211,-130.322,174.308,43.166,158.513
C06149=1045.414,403.965,-130.277,174.299,43.159,158.510
C06150=1045.405,403.719,-130.232,174.291,43.152,158.508
C06151=1045.395,403.473,-130.188,174.282,43.146,158.506
C06152=1045.385,403.227,-130.143,174.274,43.139,158.503
C06153=1045.377,402.981,-130.099,174.265,43.132,158.501
C06154=1045.368,402.735,-130.055,174.256,43.126,158.499
C06155=1045.358,402.490,-130.010,174.248,43.120,158.496
C06156=1045.349,402.244,-129.966,174.239,43.113,158.494
C06157=1045.340,401.997,-129.921,174.231,43.106,158.492
C06158=1045.331,401.752,-129.878,174.222,43.100,158.489
C06159=1045.322,401.506,-129.833,174.214,43.094,158.487
C06160=1045.312,401.260,-129.789,174.206,43.088,158.485
C06161=1045.303,401.015,-129.745,174.198,43.081,158.482
C06162=1045.294,400.769,-129.701,174.189,43.075,158.480
C06163=1045.285,400.523,-129.657,174.181,43.068,158.478
C06164=1045.276,400.277,-129.613,174.172,43.062,158.476
C06165=1045.266,400.031,-129.569,174.164,43.056,158.473
C06166=1045.257,399.784,-129.525,174.156,43.050,158.471
C06167=1045.248,399.539,-129.482,174.148,43.043,158.469
C06168=1045.239,399.293,-129.438,174.140,43.037,158.467
C06169=1045.230,399.047,-129.394,174.131,43.031,158.464
C06170=1045.221,398.801,-129.350,174.123,43.025,158.462
C06171=1045.212,398.555,-129.307,174.115,43.018,158.460
C06172=1045.203,398.309,-129.263,174.106,43.012,158.458
C06173=1045.194,398.064,-129.219,174.099,43.006,158.456
C06174=1045.185,397.817,-129.175,174.091,43.000,158.453
C06175=1045.176,397.571,-129.132,174.082,42.994,158.451
C06176=1045.167,397.326,-129.088,174.074,42.988,158.449
C06177=1045.158,397.079,-129.045,174.067,42.981,158.447
C06178=1045.150,396.834,-129.001,174.058,42.976,158.445
C06179=1045.141,396.588,-128.958,174.050,42.969,158.443
C06180=1045.132,396.342,-128.914,174.042,42.963,158.441
C06181=1045.123,396.095,-128.871,174.035,42.957,158.438
C06182=1045.114,395.850,-128.827,174.026,42.952,158.436
C06183=1045.106,395.604,-128.784,174.018,42.945,158.434
C06184=1045.096,395.358,-128.741,174.011,42.939,158.432
C06185=1045.087,395.111,-128.698,174.003,42.933,158.430
C06186=1045.079,394.866,-128.654,173.994,42.927,158.428
C06187=1045.070,394.619,-128.611,173.987,42.921,158.426
C06188=1045.061,394.373,-128.568,173.979,42.915,158.424
C06189=1045.052,394.128,-128.525,173.972,42.909,158.422
C06190=1045.043,393.881,-128.482,173.964,42.904,158.419
C06191=1045.035,393.635,-128.439,173.956,42.898,158.418
C06192=1045.026,393.389,-128.396,173.948,42.892,158.415
C06193=1045.016,393.143,-128.354,173.940,42.886,158.413
C06194=1045.008,392.897,-128.311,173.933,42.880,158.411
C06195=1044.999,392.651,-128.268,173.925,42.874,158.409
C06196=1044.990,392.405,-128.225,173.918,42.869,158.407
C06197=1044.980,392.106,-128.173,173.909,42.862,158.405
C06198=1044.970,391.806,-128.121,173.899,42.855,158.402
C06199=1044.959,391.507,-128.068,173.889,42.848,158.400
C06200=1044.948,391.207,-128.017,173.880,42.841,158.397
C06201=1044.936,390.874,-127.959,173.870,42.834,158.395
C06202=1044.924,390.539,-127.901,173.860,42.825,158.392
C06203=1044.913,390.205,-127.844,173.850,42.818,158.389
C06204=1044.901,389.872,-127.786,173.840,42.810,158.387
C06205=1044.893,389.626,-127.744,173.832,42.805,158.385
C06206=1044.884,389.379,-127.702,173.825,42.799,158.383
C06207=1044.876,389.133,-127.659,173.818,42.794,158.381
C06208=1044.867,388.887,-127.617,173.810,42.788,158.379
C06209=1044.858,388.641,-127.574,173.803,42.782,158.377
C06210=1044.849,388.394,-127.533,173.795,42.777,158.375
C06211=1044.841,388.148,-127.490,173.788,42.772,158.373
C06212=1044.832,387.902,-127.448,173.781,42.766,158.371
C06213=1044.823,387.656,-127.406,173.773,42.761,158.369
C06214=1044.815,387.410,-127.364,173.766,42.755,158.367
C06215=1044.806,387.163,-127.323,173.758,42.750,158.366
C06216=1044.797,386.917,-127.281,173.752,42.744,158.364
C06217=1044.789,386.670,-127.239,173.745,42.739,158.362
C06218=1044.780,386.424,-127.197,173.738,42.734,158.360
C06219=1044.772,386.178,-127.155,173.730,42.728,158.358
C06220=1044.763,385.932,-127.112,173.723,42.723,158.356
C06221=1044.755,385.685,-127.071,173.715,42.717,158.354
C06222=1044.746,385.439,-127.030,173.708,42.713,158.353
C06223=1044.738,385.193,-126.988,173.701,42.707,158.351
C06224=1044.729,384.946,-126.946,173.695,42.701,158.349
C06225=1044.720,384.700,-126.904,173.687,42.697,158.347
C06226=1044.712,384.454,-126.863,173.680,42.691,158.345
C06227=1044.704,384.208,-126.821,173.673,42.686,158.344
C06228=1044.696,383.962,-126.779,173.666,42.681,158.342
C06229=1044.687,383.715,-126.738,173.660,42.676,158.340
C06230=1044.678,383.469,-126.697,173.652,42.670,158.338
C06231=1044.670,383.223,-126.655,173.645,42.665,158.336
C06232=1044.662,382.976,-126.614,173.638,42.660,158.334
C06233=1044.653,382.730,-126.572,173.632,42.655,158.333
C06234=1044.645,382.483,-126.530,173.624,42.649,158.331
C06235=1044.637,382.237,-126.489,173.617,42.644,158.329
C06236=1044.628,381.991,-126.448,173.611,42.639,158.327
C06237=1044.620,381.744,-126.407,173.604,42.634,158.326
C06238=1044.612,381.498,-126.365,173.597,42.629,158.324
C06239=1044.604,381.251,-126.324,173.589,42.624,158.322
C06240=1044.595,381.005,-126.282,173.583,42.619,158.320
C06241=1044.587,380.759,-126.242,173.576,42.614,158.319
C06242=1044.579,380.512,-126.199,173.569,42.608,158.317
C06243=1044.571,380.266,-126.159,173.563,42.603,158.315
C06244=1044.563,380.020,-126.118,173.556,42.598,158.313
C06245=1044.554,379.773,-126.076,173.550,42.593,158.312
C06246=1044.547,379.527,-126.035,173.542,42.588,158.310
C06247=1044.539,379.280,-125.995,173.535,42.583,158.308
C06248=1044.530,379.033,-125.954,173.529,42.578,158.307
C06249=1044.522,378.788,-125.912,173.522,42.573,158.305
C06250=1044.514,378.541,-125.872,173.516,42.568,158.303
C06251=1044.505,378.294,-125.831,173.509,42.564,158.302
C06252=1044.497,378.048,-125.790,173.502,42.559,158.300
C06253=1044.488,377.802,-125.750,173.496,42.554,158.298
C06254=1044.480,377.555,-125.709,173.489,42.549,158.296
C06255=1044.472,377.309,-125.668,173.483,42.544,158.295
C06256=1044.463,377.063,-125.628,173.476,42.539,158.293
C06257=1044.452,376.708,-125.569,173.467,42.532,158.291
C06258=1044.440,376.354,-125.511,173.457,42.525,158.288
C06259=1044.428,376.000,-125.453,173.448,42.518,158.286
C06260=1044.417,375.647,-125.395,173.438,42.512,158.284
C06261=1044.408,375.400,-125.354,173.432,42.507,158.282
C06262=1044.400,375.153,-125.314,173.425,42.502,158.281
C06263=1044.392,374.907,-125.273,173.419,42.497,158.279
C06264=1044.384,374.660,-125.234,173.412,42.493,158.277
C06265=1044.376,374.414,-125.193,173.406,42.488,158.276
C06266=1044.368,374.167,-125.153,173.399,42.483,158.274
C06267=1044.360,373.921,-125.112,173.393,42.478,158.272
C06268=1044.351,373.674,-125.071,173.386,42.474,158.271
C06269=1044.344,373.427,-125.032,173.380,42.469,158.269
C06270=1044.336,373.181,-124.991,173.373,42.464,158.268
C06271=1044.328,372.934,-124.951,173.368,42.460,158.266
C06272=1044.319,372.688,-124.911,173.362,42.455,158.265
C06273=1044.311,372.441,-124.871,173.355,42.451,158.263
C06274=1044.303,372.195,-124.830,173.349,42.446,158.261
C06275=1044.296,371.948,-124.790,173.342,42.441,158.260
C06276=1044.288,371.701,-124.751,173.336,42.437,158.258
C06277=1044.280,371.455,-124.710,173.330,42.432,158.257
C06278=1044.272,371.208,-124.670,173.323,42.428,158.255
C06279=1044.264,370.961,-124.631,173.317,42.423,158.254
C06280=1044.256,370.714,-124.591,173.311,42.419,158.252
C06281=1044.248,370.468,-124.550,173.305,42.414,158.251
C06282=1044.240,370.222,-124.511,173.299,42.410,158.249
C06283=1044.232,369.975,-124.471,173.293,42.405,158.248
C06284=1044.224,369.729,-124.432,173.286,42.401,158.246
C06285=1044.216,369.482,-124.392,173.280,42.396,158.245
C06286=1044.208,369.235,-124.353,173.274,42.391,158.243
C06287=1044.200,368.988,-124.313,173.267,42.387,158.241
C06288=1044.192,368.741,-124.273,173.262,42.383,158.240
C06289=1044.184,368.495,-124.234,173.256,42.378,158.239
C06290=1044.176,368.248,-124.194,173.249,42.374,158.237
C06291=1044.168,368.001,-124.154,173.243,42.369,158.236
C06292=1044.161,367.755,-124.115,173.238,42.365,158.234
C06293=1044.153,367.508,-124.076,173.232,42.361,158.233
C06294=1044.145,367.261,-124.036,173.225,42.356,158.231
C06295=1044.136,367.014,-123.997,173.219,42.352,158.230
C06296=1044.129,366.767,-123.957,173.213,42.348,158.228
C06297=1044.121,366.521,-123.918,173.208,42.343,158.227
C06298=1044.113,366.274,-123.879,173.201,42.339,158.225
C06299=1044.105,366.027,-123.839,173.195,42.335,158.224
C06300=1044.097,365.780,-123.800,173.189,42.331,158.223
C06301=1044.090,365.534,-123.761,173.184,42.326,158.221
C06302=1044.082,365.287,-123.721,173.178,42.321,158.219
C06303=1044.073,365.040,-123.682,173.171,42.318,158.218
C06304=1044.067,364.794,-123.643,173.165,42.314,158.217
C06305=1044.058,364.547,-123.604,173.160,42.309,158.215
C06306=1044.051,364.299,-123.565,173.154,42.305,158.214
C06307=1044.043,364.054,-123.526,173.148,42.300,158.212
C06308=1044.035,363.806,-123.487,173.143,42.296,158.211
C06309=1044.027,363.559,-123.447,173.136,42.292,158.210
C06310=1044.020,363.313,-123.408,173.130,42.288,158.208
C06311=1044.012,363.066,-123.369,173.124,42.284,158.207
C06312=1044.005,362.819,-123.330,173.119,42.279,158.205
C06313=1043.994,362.484,-123.278,173.111,42.273,158.203
C06314=1043.984,362.150,-123.225,173.103,42.268,158.202
C06315=1043.973,361.816,-123.173,173.095,42.262,158.200
C06316=1043.962,361.481,-123.120,173.088,42.257,158.198
C06317=1043.954,361.235,-123.081,173.082,42.253,158.197
C06318=1043.947,360.988,-123.042,173.076,42.249,158.195
C06319=1043.939,360.741,-123.004,173.071,42.245,158.194
C06320=1043.931,360.494,-122.965,173.064,42.241,158.192
C06321=1043.924,360.247,-122.927,173.059,42.237,158.191
C06322=1043.916,360.000,-122.888,173.053,42.233,158.190
C06323=1043.909,359.753,-122.849,173.047,42.229,158.188
C06324=1043.901,359.506,-122.811,173.042,42.225,158.187
C06325=1043.893,359.260,-122.772,173.036,42.221,158.186
C06326=1043.885,359.012,-122.734,173.030,42.217,158.184
C06327=1043.877,358.766,-122.696,173.025,42.212,158.183
C06328=1043.870,358.519,-122.657,173.019,42.208,158.182
C06329=1043.862,358.272,-122.618,173.014,42.204,158.180
C06330=1043.855,358.025,-122.580,173.008,42.200,158.179
C06331=1043.847,357.778,-122.541,173.003,42.197,158.178
C06332=1043.839,357.532,-122.503,172.997,42.193,158.177
C06333=1043.832,357.285,-122.465,172.991,42.189,158.175
C06334=1043.824,357.037,-122.427,172.986,42.185,158.174
C06335=1043.816,356.791,-122.389,172.980,42.181,158.172
C06336=1043.809,356.544,-122.350,172.975,42.177,158.171
C06337=1043.801,356.296,-122.312,172.969,42.173,158.170
C06338=1043.793,356.050,-122.274,172.963,42.169,158.169
C06339=1043.786,355.803,-122.236,172.958,42.165,158.167
C06340=1043.778,355.556,-122.198,172.952,42.161,158.166
C06341=1043.770,355.309,-122.160,172.947,42.158,158.165
C06342=1043.763,355.062,-122.122,172.941,42.154,158.164
C06343=1043.755,354.815,-122.084,172.936,42.150,158.162
C06344=1043.748,354.568,-122.046,172.930,42.146,158.161
C06345=1043.740,354.321,-122.008,172.926,42.142,158.160
C06346=1043.733,354.074,-121.970,172.920,42.139,158.159
C06347=1043.725,353.827,-121.932,172.915,42.134,158.157
C06348=1043.717,353.580,-121.894,172.909,42.131,158.156
C06349=1043.710,353.333,-121.856,172.904,42.127,158.155
C06350=1043.703,353.086,-121.818,172.898,42.123,158.154
C06351=1043.695,352.839,-121.781,172.893,42.120,158.152
C06352=1043.687,352.592,-121.742,172.887,42.116,158.151
C06353=1043.680,352.344,-121.705,172.882,42.112,158.150
C06354=1043.672,352.098,-121.668,172.877,42.108,158.149
C06355=1043.665,351.851,-121.630,172.872,42.105,158.147
C06356=1043.657,351.604,-121.592,172.867,42.101,158.146
C06357=1043.650,351.357,-121.555,172.861,42.097,158.145
C06358=1043.643,351.110,-121.517,172.856,42.093,158.144
C06359=1043.635,350.862,-121.479,172.850,42.090,158.142
C06360=1043.627,350.615,-121.441,172.846,42.086,158.141
C06361=1043.620,350.368,-121.403,172.840,42.082,158.140
C06362=1043.613,350.121,-121.366,172.835,42.079,158.139
C06363=1043.605,349.874,-121.329,172.829,42.075,158.138
C06364=1043.598,349.627,-121.291,172.824,42.072,158.136
C06365=1043.590,349.380,-121.254,172.819,42.068,158.135
C06366=1043.582,349.133,-121.217,172.814,42.065,158.134
C06367=1043.575,348.886,-121.179,172.809,42.060,158.133
C06368=1043.568,348.639,-121.142,172.803,42.057,158.132
C06369=1043.558,348.310,-121.093,172.796,42.052,158.130
C06370=1043.548,347.982,-121.042,172.790,42.048,158.129
C06371=1043.538,347.653,-120.994,172.783,42.043,158.127
C06372=1043.528,347.325,-120.944,172.776,42.038,158.125
C06373=1043.521,347.077,-120.907,172.771,42.035,158.124
C06374=1043.513,346.830,-120.869,172.766,42.031,158.123
C06375=1043.506,346.583,-120.833,172.761,42.027,158.122
C06376=1043.499,346.336,-120.795,172.755,42.024,158.121
C06377=1043.491,346.089,-120.758,172.750,42.020,158.120
C06378=1043.483,345.842,-120.721,172.746,42.017,158.118
C06379=1043.476,345.594,-120.684,172.740,42.013,158.117
C06380=1043.468,345.347,-120.647,172.735,42.010,158.116
C06381=1043.462,345.101,-120.610,172.730,42.007,158.115
C06382=1043.455,344.853,-120.573,172.725,42.003,158.114
C06383=1043.447,344.606,-120.536,172.720,42.000,158.113
C06384=1043.440,344.358,-120.499,172.715,41.996,158.112
C06385=1043.432,344.112,-120.463,172.710,41.993,158.111
C06386=1043.425,343.864,-120.426,172.705,41.989,158.109
C06387=1043.417,343.617,-120.389,172.700,41.986,158.108
C06388=1043.411,343.370,-120.352,172.695,41.982,158.107
C06389=1043.403,343.123,-120.315,172.690,41.979,158.106
C06390=1043.396,342.875,-120.279,172.685,41.976,158.105
C06391=1043.388,342.628,-120.241,172.680,41.972,158.104
C06392=1043.381,342.381,-120.205,172.675,41.968,158.103
C06393=1043.374,342.134,-120.168,172.671,41.965,158.102
C06394=1043.366,341.887,-120.132,172.665,41.962,158.100
C06395=1043.359,341.639,-120.095,172.660,41.959,158.099
C06396=1043.352,341.392,-120.058,172.656,41.955,158.098
C06397=1043.344,341.146,-120.022,172.650,41.952,158.097
C06398=1043.337,340.898,-119.986,172.645,41.949,158.096
C06399=1043.330,340.650,-119.949,172.641,41.945,158.095
C06400=1043.322,340.403,-119.913,172.636,41.942,158.094
C06401=1043.315,340.156,-119.877,172.630,41.938,158.093
C06402=1043.308,339.909,-119.839,172.626,41.935,158.092
C06403=1043.300,339.662,-119.803,172.621,41.932,158.091
C06404=1043.293,339.414,-119.767,172.617,41.929,158.090
C06405=1043.286,339.167,-119.730,172.611,41.926,158.089
C06406=1043.279,338.920,-119.694,172.607,41.922,158.088
C06407=1043.271,338.672,-119.658,172.602,41.919,158.087
C06408=1043.264,338.425,-119.622,172.597,41.916,158.085
C06409=1043.257,338.178,-119.585,172.592,41.912,158.084
C06410=1043.250,337.931,-119.549,172.587,41.909,158.083
C06411=1043.242,337.684,-119.513,172.583,41.906,158.082
C06412=1043.235,337.436,-119.476,172.578,41.903,158.081
C06413=1043.228,337.189,-119.441,172.573,41.900,158.080
C06414=1043.220,336.942,-119.404,172.568,41.896,158.079
C06415=1043.213,336.695,-119.369,172.564,41.893,158.078
C06416=1043.206,336.447,-119.332,172.559,41.890,158.077
C06417=1043.199,336.200,-119.295,172.554,41.886,158.076
C06418=1043.192,335.953,-119.260,172.549,41.883,158.075
C06419=1043.184,335.705,-119.224,172.545,41.880,158.074
C06420=1043.178,335.458,-119.188,172.540,41.877,158.073
C06421=1043.170,335.210,-119.151,172.536,41.874,158.072
C06422=1043.163,334.964,-119.116,172.530,41.871,158.071
C06423=1043.156,334.715,-119.080,172.526,41.867,158.070
C06424=1043.149,334.469,-119.044,172.521,41.864,158.069
C06425=1043.139,334.137,-118.996,172.515,41.860,158.067
C06426=1043.129,333.804,-118.948,172.509,41.856,158.066
C06427=1043.119,333.472,-118.900,172.502,41.852,158.065
C06428=1043.110,333.139,-118.852,172.496,41.848,158.063
C06429=1043.102,332.892,-118.816,172.492,41.845,158.062
C06430=1043.095,332.645,-118.780,172.487,41.842,158.061
C06431=1043.088,332.398,-118.745,172.482,41.838,158.060
C06432=1043.080,332.150,-118.709,172.478,41.835,158.059
C06433=1043.074,331.903,-118.674,172.473,41.832,158.058
C06434=1043.066,331.655,-118.638,172.469,41.830,158.058
C06435=1043.059,331.408,-118.603,172.464,41.827,158.057
C06436=1043.052,331.161,-118.567,172.460,41.824,158.056
C06437=1043.045,330.913,-118.531,172.454,41.821,158.055
C06438=1043.038,330.666,-118.496,172.450,41.818,158.054
C06439=1043.030,330.418,-118.460,172.446,41.814,158.053
C06440=1043.024,330.171,-118.425,172.441,41.811,158.052
C06441=1043.017,329.924,-118.390,172.437,41.808,158.051
C06442=1043.009,329.676,-118.353,172.432,41.805,158.050
C06443=1043.002,329.429,-118.318,172.427,41.802,158.049
C06444=1042.996,329.182,-118.283,172.423,41.799,158.048
C06445=1042.988,328.933,-118.248,172.418,41.797,158.047
C06446=1042.981,328.687,-118.212,172.414,41.793,158.046
C06447=1042.974,328.440,-118.177,172.409,41.790,158.045
C06448=1042.966,328.192,-118.142,172.405,41.787,158.044
C06449=1042.959,327.945,-118.107,172.401,41.785,158.043
C06450=1042.952,327.697,-118.072,172.396,41.782,158.042
C06451=1042.945,327.449,-118.037,172.392,41.779,158.041
C06452=1042.937,327.202,-118.002,172.387,41.776,158.040
C06453=1042.930,326.955,-117.967,172.383,41.773,158.039
C06454=1042.922,326.707,-117.932,172.379,41.771,158.038
C06455=1042.916,326.460,-117.897,172.373,41.768,158.037
C06456=1042.909,326.212,-117.862,172.369,41.764,158.036
C06457=1042.901,325.965,-117.827,172.365,41.762,158.036
C06458=1042.894,325.717,-117.792,172.360,41.759,158.035
C06459=1042.886,325.470,-117.757,172.356,41.756,158.034
C06460=1042.880,325.223,-117.722,172.352,41.753,158.033
C06461=1042.873,324.975,-117.687,172.347,41.751,158.032
C06462=1042.865,324.727,-117.653,172.343,41.748,158.031
C06463=1042.858,324.480,-117.618,172.339,41.745,158.030
C06464=1042.851,324.233,-117.583,172.334,41.742,158.029
C06465=1042.844,323.985,-117.548,172.330,41.739,158.028
C06466=1042.836,323.738,-117.513,172.326,41.736,158.027
C06467=1042.830,323.491,-117.478,172.321,41.734,158.026
C06468=1042.822,323.242,-117.444,172.317,41.731,158.025
C06469=1042.815,322.995,-117.409,172.313,41.728,158.025
C06470=1042.808,322.748,-117.374,172.309,41.725,158.024
C06471=1042.801,322.501,-117.339,172.304,41.723,158.023
C06472=1042.794,322.253,-117.305,172.299,41.720,158.022
C06473=1042.787,322.006,-117.270,172.295,41.717,158.021
C06474=1042.780,321.758,-117.235,172.291,41.714,158.020
C06475=1042.773,321.511,-117.201,172.286,41.711,158.019
C06476=1042.766,321.263,-117.166,172.282,41.709,158.018
C06477=1042.759,321.016,-117.132,172.278,41.706,158.017
C06478=1042.752,320.767,-117.097,172.274,41.703,158.017
C06479=1042.744,320.520,-117.062,172.269,41.700,158.016
C06480=1042.738,320.272,-117.028,172.265,41.698,158.015
C06481=1042.728,319.936,-116.981,172.260,41.694,158.014
C06482=1042.719,319.599,-116.934,172.253,41.690,158.012
C06483=1042.709,319.261,-116.887,172.248,41.686,158.011
C06484=1042.700,318.924,-116.840,172.243,41.683,158.010
C06485=1042.693,318.677,-116.805,172.238,41.680,158.009
C06486=1042.686,318.429,-116.771,172.234,41.677,158.008
C06487=1042.679,318.182,-116.736,172.230,41.674,158.007
C06488=1042.672,317.934,-116.702,172.226,41.672,158.007
C06489=1042.665,317.686,-116.668,172.222,41.669,158.006
C06490=1042.658,317.439,-116.633,172.218,41.666,158.005
C06491=1042.652,317.192,-116.599,172.213,41.664,158.004
C06492=1042.644,316.945,-116.565,172.209,41.661,158.003
C06493=1042.638,316.697,-116.530,172.205,41.658,158.002
C06494=1042.631,316.449,-116.497,172.201,41.655,158.001
C06495=1042.624,316.202,-116.461,172.197,41.653,158.000
C06496=1042.617,315.954,-116.428,172.193,41.650,158.000
C06497=1042.610,315.706,-116.393,172.189,41.647,157.999
C06498=1042.604,315.459,-116.360,172.184,41.645,157.998
C06499=1042.597,315.212,-116.325,172.180,41.642,157.997
C06500=1042.590,314.964,-116.291,172.176,41.639,157.996
C06501=1042.583,314.716,-116.256,172.172,41.637,157.995
C06502=1042.576,314.469,-116.223,172.168,41.634,157.994
C06503=1042.570,314.221,-116.189,172.164,41.631,157.994
C06504=1042.563,313.974,-116.154,172.160,41.629,157.993
C06505=1042.556,313.726,-116.120,172.156,41.626,157.992
C06506=1042.549,313.479,-116.086,172.152,41.623,157.991
C06507=1042.542,313.232,-116.052,172.148,41.621,157.990
C06508=1042.536,312.984,-116.018,172.143,41.618,157.989
C06509=1042.529,312.736,-115.984,172.139,41.615,157.988
C06510=1042.523,312.489,-115.950,172.135,41.613,157.988
C06511=1042.516,312.241,-115.916,172.131,41.610,157.987
C06512=1042.508,311.993,-115.882,172.127,41.607,157.986
C06513=1042.501,311.746,-115.849,172.123,41.605,157.985
C06514=1042.494,311.498,-115.815,172.119,41.603,157.985
C06515=1042.487,311.251,-115.781,172.116,41.600,157.984
C06516=1042.480,311.003,-115.748,172.112,41.598,157.983
C06517=1042.473,310.755,-115.715,172.108,41.595,157.982
C06518=1042.465,310.508,-115.681,172.103,41.593,157.981
C06519=1042.458,310.260,-115.647,172.099,41.590,157.980
C06520=1042.452,310.013,-115.614,172.095,41.588,157.980
C06521=1042.445,309.765,-115.581,172.091,41.585,157.979
C06522=1042.437,309.517,-115.547,172.087,41.583,157.978
C06523=1042.431,309.270,-115.513,172.083,41.580,157.977
C06524=1042.424,309.022,-115.480,172.079,41.578,157.977
C06525=1042.416,308.774,-115.447,172.076,41.576,157.976
C06526=1042.409,308.527,-115.413,172.072,41.573,157.975
C06527=1042.403,308.279,-115.380,172.068,41.571,157.974
C06528=1042.395,308.032,-115.347,172.064,41.568,157.973
C06529=1042.389,307.785,-115.313,172.060,41.566,157.973
C06530=1042.382,307.536,-115.280,172.056,41.563,157.972
C06531=1042.375,307.289,-115.246,172.052,41.561,157.971
C06532=1042.367,307.042,-115.213,172.048,41.558,157.970
C06533=1042.360,306.794,-115.180,172.044,41.556,157.970
C06534=1042.353,306.546,-115.146,172.039,41.554,157.969
C06535=1042.347,306.298,-115.114,172.036,41.551,157.968
C06536=1042.340,306.051,-115.080,172.032,41.549,157.967
C06537=1042.331,305.718,-115.035,172.026,41.546,157.966
C06538=1042.321,305.386,-114.991,172.021,41.542,157.965
C06539=1042.312,305.053,-114.947,172.016,41.539,157.964
C06540=1042.302,304.721,-114.902,172.011,41.536,157.963
C06541=1042.296,304.474,-114.869,172.007,41.534,157.962
C06542=1042.289,304.225,-114.836,172.003,41.531,157.962
C06543=1042.283,303.978,-114.803,171.999,41.529,157.961
C06544=1042.275,303.730,-114.769,171.997,41.526,157.960
C06545=1042.269,303.483,-114.736,171.993,41.524,157.959
C06546=1042.262,303.235,-114.704,171.989,41.521,157.959
C06547=1042.255,302.988,-114.670,171.985,41.519,157.958
C06548=1042.248,302.739,-114.637,171.981,41.517,157.957
C06549=1042.242,302.492,-114.605,171.977,41.514,157.956
C06550=1042.235,302.244,-114.571,171.973,41.512,157.956
C06551=1042.228,301.997,-114.539,171.969,41.509,157.955
C06552=1042.221,301.749,-114.506,171.966,41.507,157.954
C06553=1042.214,301.502,-114.472,171.962,41.505,157.953
C06554=1042.208,301.254,-114.439,171.958,41.502,157.952
C06555=1042.201,301.006,-114.406,171.954,41.500,157.952
C06556=1042.194,300.758,-114.374,171.950,41.498,157.951
C06557=1042.187,300.510,-114.341,171.946,41.496,157.950
C06558=1042.181,300.263,-114.308,171.944,41.493,157.950
C06559=1042.174,300.016,-114.275,171.940,41.490,157.949
C06560=1042.167,299.767,-114.242,171.936,41.488,157.948
C06561=1042.160,299.520,-114.210,171.932,41.486,157.947
C06562=1042.153,299.272,-114.176,171.928,41.484,157.947
C06563=1042.147,299.024,-114.144,171.924,41.481,157.946
C06564=1042.141,298.776,-114.111,171.920,41.479,157.945
C06565=1042.134,298.528,-114.078,171.917,41.476,157.944
C06566=1042.127,298.281,-114.046,171.914,41.474,157.944
C06567=1042.120,298.033,-114.013,171.910,41.472,157.943
C06568=1042.114,297.786,-113.980,171.906,41.470,157.942
C06569=1042.107,297.537,-113.947,171.902,41.467,157.941
C06570=1042.100,297.290,-113.915,171.899,41.465,157.941
C06571=1042.094,297.043,-113.882,171.895,41.462,157.940
C06572=1042.087,296.794,-113.849,171.892,41.460,157.939
C06573=1042.081,296.547,-113.816,171.888,41.458,157.938
C06574=1042.074,296.299,-113.784,171.884,41.456,157.938
C06575=1042.067,296.052,-113.751,171.880,41.453,157.937
C06576=1042.060,295.803,-113.718,171.877,41.451,157.936
C06577=1042.054,295.556,-113.686,171.873,41.448,157.936
C06578=1042.047,295.309,-113.653,171.870,41.446,157.935
C06579=1042.041,295.060,-113.621,171.866,41.444,157.934
C06580=1042.034,294.812,-113.589,171.862,41.442,157.933
C06581=1042.027,294.565,-113.556,171.858,41.439,157.933
C06582=1042.020,294.318,-113.524,171.855,41.437,157.932
C06583=1042.014,294.069,-113.492,171.852,41.435,157.931
C06584=1042.007,293.821,-113.459,171.848,41.433,157.931
C06585=1042.000,293.574,-113.427,171.844,41.431,157.930
C06586=1041.994,293.326,-113.395,171.840,41.428,157.929
C06587=1041.987,293.079,-113.363,171.837,41.426,157.929
C06588=1041.980,292.830,-113.330,171.833,41.424,157.928
C06589=1041.973,292.582,-113.299,171.830,41.422,157.927
C06590=1041.966,292.335,-113.266,171.826,41.419,157.926
C06591=1041.960,292.087,-113.234,171.823,41.417,157.926
C06592=1041.952,291.839,-113.202,171.819,41.415,157.925
C06593=1041.944,291.523,-113.161,171.815,41.413,157.924
C06594=1041.935,291.207,-113.121,171.810,41.409,157.923
C06595=1041.926,290.891,-113.079,171.806,41.407,157.923
C06596=1041.918,290.575,-113.038,171.801,41.404,157.922
C06597=1041.911,290.327,-113.007,171.797,41.402,157.921
C06598=1041.904,290.080,-112.974,171.794,41.400,157.920
C06599=1041.898,289.832,-112.942,171.791,41.398,157.920
C06600=1041.891,289.584,-112.911,171.787,41.396,157.919
C06601=1041.884,289.336,-112.878,171.783,41.393,157.918
C06602=1041.877,289.088,-112.847,171.780,41.391,157.918
C06603=1041.871,288.841,-112.814,171.776,41.389,157.917
C06604=1041.864,288.593,-112.783,171.773,41.387,157.916
C06605=1041.857,288.345,-112.751,171.769,41.385,157.916
C06606=1041.850,288.098,-112.719,171.766,41.383,157.915
C06607=1041.844,287.849,-112.687,171.763,41.380,157.914
C06608=1041.838,287.601,-112.656,171.759,41.378,157.914
C06609=1041.831,287.354,-112.624,171.756,41.376,157.913
C06610=1041.823,287.106,-112.592,171.752,41.374,157.912
C06611=1041.817,286.858,-112.560,171.748,41.372,157.912
C06612=1041.810,286.610,-112.529,171.745,41.370,157.911
C06613=1041.803,286.362,-112.498,171.742,41.367,157.910
C06614=1041.796,286.115,-112.465,171.738,41.365,157.910
C06615=1041.789,285.867,-112.434,171.735,41.363,157.909
C06616=1041.783,285.619,-112.403,171.732,41.361,157.908
C06617=1041.777,285.371,-112.371,171.728,41.359,157.908
C06618=1041.770,285.123,-112.339,171.724,41.357,157.907
C06619=1041.763,284.875,-112.308,171.721,41.355,157.906
C06620=1041.756,284.627,-112.276,171.718,41.353,157.906
C06621=1041.750,284.379,-112.245,171.714,41.351,157.905
C06622=1041.743,284.131,-112.213,171.710,41.349,157.904
C06623=1041.736,283.883,-112.182,171.708,41.347,157.904
C06624=1041.730,283.635,-112.150,171.704,41.345,157.903
C06625=1041.723,283.387,-112.119,171.700,41.343,157.902
C06626=1041.716,283.139,-112.088,171.698,41.340,157.902
C06627=1041.709,282.891,-112.056,171.694,41.338,157.901
C06628=1041.703,282.644,-112.025,171.690,41.336,157.900
C06629=1041.696,282.396,-111.993,171.687,41.334,157.900
C06630=1041.689,282.148,-111.962,171.684,41.332,157.899
C06631=1041.682,281.900,-111.930,171.680,41.330,157.899
C06632=1041.676,281.652,-111.899,171.677,41.328,157.898
C06633=1041.669,281.404,-111.868,171.673,41.326,157.897
C06634=1041.662,281.156,-111.836,171.671,41.324,157.897
C06635=1041.656,280.908,-111.805,171.667,41.322,157.896
C06636=1041.649,280.660,-111.773,171.663,41.320,157.895
C06637=1041.642,280.412,-111.742,171.661,41.318,157.895
C06638=1041.635,280.165,-111.710,171.657,41.316,157.894
C06639=1041.629,279.916,-111.680,171.654,41.314,157.894
C06640=1041.622,279.668,-111.648,171.651,41.312,157.893
C06641=1041.615,279.420,-111.617,171.647,41.310,157.892
C06642=1041.609,279.173,-111.586,171.644,41.308,157.892
C06643=1041.603,278.925,-111.554,171.640,41.306,157.891
C06644=1041.595,278.677,-111.524,171.638,41.303,157.890
C06645=1041.589,278.429,-111.493,171.634,41.301,157.890
C06646=1041.582,278.181,-111.461,171.630,41.300,157.889
C06647=1041.576,277.933,-111.431,171.628,41.298,157.889
C06648=1041.569,277.685,-111.399,171.624,41.296,157.888
C06649=1041.560,277.381,-111.362,171.620,41.293,157.887
C06650=1041.552,277.076,-111.323,171.616,41.291,157.886
C06651=1041.544,276.773,-111.285,171.612,41.288,157.886
C06652=1041.536,276.468,-111.248,171.609,41.286,157.885
C06653=1041.529,276.221,-111.217,171.605,41.284,157.884
C06654=1041.522,275.972,-111.186,171.601,41.282,157.884
C06655=1041.516,275.724,-111.155,171.599,41.280,157.883
C06656=1041.509,275.476,-111.123,171.595,41.278,157.882
C06657=1041.502,275.229,-111.094,171.592,41.276,157.882
C06658=1041.496,274.981,-111.062,171.588,41.274,157.881
C06659=1041.489,274.732,-111.032,171.586,41.272,157.881
C06660=1041.482,274.484,-111.000,171.582,41.270,157.880
C06661=1041.475,274.236,-110.970,171.579,41.268,157.879
C06662=1041.469,273.989,-110.939,171.576,41.266,157.879
C06663=1041.463,273.740,-110.908,171.572,41.265,157.878
C06664=1041.456,273.492,-110.878,171.569,41.262,157.878
C06665=1041.449,273.244,-110.847,171.566,41.260,157.877
C06666=1041.442,272.996,-110.816,171.563,41.258,157.876
C06667=1041.436,272.749,-110.785,171.559,41.257,157.876
C06668=1041.429,272.500,-110.755,171.557,41.255,157.875
C06669=1041.422,272.252,-110.725,171.553,41.252,157.875
C06670=1041.415,272.004,-110.693,171.550,41.251,157.874
C06671=1041.409,271.756,-110.663,171.547,41.249,157.873
C06672=1041.402,271.508,-110.633,171.544,41.247,157.873
C06673=1041.396,271.260,-110.601,171.540,41.245,157.872
C06674=1041.388,271.012,-110.571,171.538,41.243,157.872
C06675=1041.383,270.764,-110.541,171.534,41.241,157.871
C06676=1041.375,270.516,-110.511,171.531,41.239,157.870
C06677=1041.369,270.268,-110.480,171.528,41.237,157.870
C06678=1041.362,270.020,-110.449,171.525,41.235,157.869
C06679=1041.356,269.772,-110.419,171.521,41.233,157.869
C06680=1041.349,269.524,-110.389,171.519,41.232,157.868
C06681=1041.342,269.275,-110.358,171.515,41.229,157.867
C06682=1041.336,269.028,-110.328,171.512,41.227,157.867
C06683=1041.329,268.779,-110.297,171.509,41.226,157.866
C06684=1041.322,268.532,-110.267,171.506,41.224,157.866
C06685=1041.316,268.284,-110.236,171.504,41.222,157.865
C06686=1041.309,268.036,-110.206,171.500,41.220,157.865
C06687=1041.302,267.787,-110.175,171.497,41.218,157.864
C06688=1041.296,267.540,-110.146,171.494,41.216,157.863
C06689=1041.289,267.291,-110.115,171.491,41.214,157.863
C06690=1041.282,267.043,-110.085,171.487,41.213,157.862
C06691=1041.276,266.795,-110.055,171.485,41.211,157.862
C06692=1041.269,266.547,-110.024,171.481,41.208,157.861
C06693=1041.262,266.299,-109.994,171.478,41.207,157.861
C06694=1041.256,266.051,-109.964,171.476,41.205,157.860
C06695=1041.249,265.803,-109.934,171.472,41.203,157.859
C06696=1041.242,265.554,-109.904,171.469,41.201,157.859
C06697=1041.235,265.307,-109.874,171.466,41.200,157.858
C06698=1041.229,265.058,-109.843,171.463,41.197,157.858
C06699=1041.222,264.811,-109.813,171.459,41.195,157.857
C06700=1041.215,264.563,-109.783,171.457,41.194,157.857
C06701=1041.209,264.314,-109.753,171.454,41.192,157.856
C06702=1041.203,264.066,-109.724,171.451,41.190,157.855
C06703=1041.195,263.818,-109.693,171.448,41.188,157.855
C06704=1041.190,263.570,-109.663,171.444,41.187,157.854
C06705=1041.181,263.270,-109.627,171.441,41.184,157.854
C06706=1041.173,262.971,-109.591,171.438,41.182,157.853
C06707=1041.165,262.671,-109.555,171.434,41.180,157.852
C06708=1041.157,262.371,-109.518,171.430,41.177,157.852
C06709=1041.151,262.123,-109.488,171.427,41.175,157.851
C06710=1041.144,261.875,-109.458,171.424,41.174,157.850
C06711=1041.137,261.628,-109.429,171.421,41.172,157.850
C06712=1041.130,261.379,-109.399,171.418,41.170,157.849
C06713=1041.123,261.130,-109.369,171.415,41.168,157.849
C06714=1041.117,260.883,-109.339,171.412,41.167,157.848
C06715=1041.110,260.634,-109.310,171.409,41.165,157.848
C06716=1041.103,260.387,-109.280,171.406,41.163,157.847
C06717=1041.096,260.138,-109.251,171.403,41.161,157.847
C06718=1041.090,259.890,-109.221,171.400,41.160,157.846
C06719=1041.082,259.642,-109.192,171.397,41.158,157.845
C06720=1041.075,259.394,-109.162,171.394,41.156,157.845
C06721=1041.068,259.146,-109.132,171.391,41.154,157.844
C06722=1041.062,258.897,-109.103,171.388,41.152,157.844
C06723=1041.055,258.650,-109.073,171.385,41.151,157.843
C06724=1041.048,258.401,-109.044,171.383,41.149,157.843
C06725=1041.042,258.153,-109.014,171.379,41.147,157.842
C06726=1041.035,257.905,-108.985,171.377,41.146,157.842
C06727=1041.029,257.656,-108.955,171.374,41.143,157.841
C06728=1041.021,257.408,-108.925,171.370,41.142,157.841
C06729=1041.015,257.160,-108.896,171.368,41.140,157.840
C06730=1041.008,256.912,-108.866,171.365,41.138,157.840
C06731=1041.002,256.664,-108.837,171.362,41.137,157.839
C06732=1040.995,256.415,-108.807,171.359,41.134,157.838
C06733=1040.988,256.168,-108.779,171.356,41.133,157.838
C06734=1040.981,255.919,-108.749,171.353,41.131,157.837
C06735=1040.974,255.671,-108.719,171.350,41.129,157.837
C06736=1040.968,255.423,-108.690,171.348,41.128,157.836
C06737=1040.961,255.175,-108.660,171.344,41.126,157.836
C06738=1040.955,254.927,-108.631,171.341,41.124,157.835
C06739=1040.948,254.678,-108.602,171.339,41.122,157.835
C06740=1040.941,254.430,-108.572,171.335,41.121,157.834
C06741=1040.935,254.182,-108.543,171.333,41.119,157.834
C06742=1040.928,253.934,-108.514,171.330,41.117,157.833
C06743=1040.921,253.686,-108.485,171.327,41.116,157.833
C06744=1040.914,253.437,-108.455,171.324,41.113,157.832
C06745=1040.908,253.189,-108.426,171.321,41.112,157.832
C06746=1040.901,252.941,-108.397,171.319,41.110,157.831
C06747=1040.895,252.692,-108.368,171.316,41.108,157.830
C06748=1040.888,252.445,-108.338,171.312,41.107,157.830
C06749=1040.882,252.197,-108.309,171.310,41.104,157.829
C06750=1040.875,251.948,-108.279,171.307,41.103,157.829
C06751=1040.869,251.700,-108.250,171.304,41.101,157.828
C06752=1040.862,251.452,-108.222,171.301,41.099,157.828
C06753=1040.854,251.204,-108.192,171.299,41.097,157.827
C06754=1040.848,250.956,-108.163,171.296,41.096,157.827
C06755=1040.842,250.707,-108.134,171.293,41.094,157.826
C06756=1040.835,250.459,-108.104,171.290,41.092,157.826
C06757=1040.829,250.211,-108.075,171.287,41.091,157.825
C06758=1040.823,249.962,-108.046,171.285,41.088,157.825
C06759=1040.816,249.714,-108.017,171.282,41.087,157.824
C06760=1040.808,249.466,-107.988,171.278,41.085,157.823
C06761=1040.801,249.165,-107.952,171.276,41.083,157.823
C06762=1040.793,248.864,-107.917,171.272,41.080,157.822
C06763=1040.785,248.563,-107.882,171.268,41.078,157.822
C06764=1040.777,248.262,-107.846,171.265,41.076,157.821
C06765=1040.771,248.014,-107.817,171.263,41.075,157.821
C06766=1040.764,247.766,-107.788,171.259,41.072,157.820
C06767=1040.758,247.518,-107.759,171.257,41.071,157.819
C06768=1040.751,247.269,-107.730,171.254,41.069,157.819
C06769=1040.745,247.021,-107.701,171.252,41.067,157.818
C06770=1040.738,246.773,-107.672,171.249,41.065,157.818
C06771=1040.732,246.525,-107.643,171.246,41.064,157.817
C06772=1040.726,246.276,-107.614,171.243,41.062,157.817
C06773=1040.719,246.028,-107.585,171.240,41.060,157.816
C06774=1040.712,245.779,-107.556,171.238,41.059,157.816
C06775=1040.707,245.531,-107.527,171.235,41.056,157.815
C06776=1040.700,245.283,-107.499,171.232,41.055,157.815
C06777=1040.693,245.035,-107.470,171.230,41.053,157.814
C06778=1040.686,244.786,-107.441,171.226,41.051,157.814
C06779=1040.679,244.538,-107.412,171.224,41.049,157.813
C06780=1040.673,244.290,-107.383,171.221,41.048,157.813
C06781=1040.667,244.041,-107.355,171.219,41.046,157.812
C06782=1040.660,243.793,-107.326,171.216,41.044,157.812
C06783=1040.653,243.545,-107.297,171.213,41.042,157.811
C06784=1040.646,243.297,-107.268,171.211,41.041,157.811
C06785=1040.640,243.048,-107.240,171.207,41.039,157.810
C06786=1040.634,242.800,-107.212,171.205,41.037,157.809
C06787=1040.627,242.552,-107.183,171.202,41.036,157.809
C06788=1040.621,242.304,-107.154,171.200,41.034,157.809
C06789=1040.614,242.055,-107.126,171.197,41.032,157.808
C06790=1040.607,241.807,-107.096,171.194,41.030,157.807
C06791=1040.600,241.559,-107.068,171.192,41.028,157.807
C06792=1040.595,241.310,-107.040,171.189,41.027,157.806
C06793=1040.588,241.062,-107.011,171.186,41.025,157.806
C06794=1040.581,240.814,-106.982,171.183,41.023,157.805
C06795=1040.575,240.566,-106.954,171.181,41.022,157.805
C06796=1040.568,240.317,-106.925,171.178,41.020,157.804
C06797=1040.561,240.068,-106.897,171.176,41.018,157.804
C06798=1040.554,239.821,-106.869,171.173,41.017,157.803
C06799=1040.548,239.572,-106.841,171.170,41.015,157.803
C06800=1040.541,239.324,-106.812,171.168,41.013,157.802
C06801=1040.534,239.076,-106.784,171.164,41.011,157.802
C06802=1040.528,238.827,-106.755,171.162,41.010,157.801
C06803=1040.521,238.579,-106.727,171.159,41.008,157.801
C06804=1040.514,238.330,-106.699,171.157,41.007,157.800
C06805=1040.508,238.082,-106.671,171.154,41.004,157.800
C06806=1040.501,237.834,-106.642,171.152,41.003,157.799
C06807=1040.494,237.585,-106.614,171.149,41.001,157.799
C06808=1040.488,237.337,-106.585,171.147,41.000,157.798
C06809=1040.481,237.089,-106.558,171.144,40.998,157.798
C06810=1040.474,236.841,-106.529,171.142,40.996,157.798
C06811=1040.468,236.593,-106.501,171.138,40.995,157.797
C06812=1040.462,236.344,-106.473,171.135,40.993,157.796
C06813=1040.455,236.096,-106.445,171.133,40.991,157.796
C06814=1040.448,235.848,-106.417,171.130,40.989,157.795
C06815=1040.441,235.599,-106.388,171.128,40.988,157.795
C06816=1040.435,235.350,-106.360,171.125,40.986,157.795
C06817=1040.426,235.044,-106.325,171.123,40.984,157.794
C06818=1040.418,234.737,-106.290,171.119,40.982,157.793
C06819=1040.410,234.430,-106.256,171.116,40.980,157.793
C06820=1040.402,234.123,-106.221,171.112,40.978,157.792
C06821=1040.395,233.874,-106.193,171.110,40.976,157.792
C06822=1040.388,233.627,-106.165,171.107,40.974,157.791
C06823=1040.382,233.378,-106.137,171.105,40.973,157.791
C06824=1040.376,233.129,-106.109,171.102,40.971,157.790
C06825=1040.369,232.881,-106.081,171.100,40.969,157.790
C06826=1040.362,232.633,-106.053,171.097,40.967,157.789
C06827=1040.356,232.384,-106.024,171.095,40.966,157.789
C06828=1040.349,232.136,-105.997,171.092,40.964,157.788
C06829=1040.343,231.888,-105.969,171.090,40.962,157.788
C06830=1040.336,231.639,-105.941,171.087,40.961,157.787
C06831=1040.329,231.391,-105.913,171.085,40.959,157.787
C06832=1040.322,231.143,-105.885,171.082,40.957,157.786
C06833=1040.316,230.894,-105.857,171.079,40.955,157.786
C06834=1040.310,230.646,-105.829,171.077,40.954,157.785
C06835=1040.304,230.398,-105.802,171.074,40.952,157.785
C06836=1040.297,230.149,-105.774,171.072,40.951,157.784
C06837=1040.290,229.901,-105.746,171.069,40.949,157.784
C06838=1040.284,229.653,-105.718,171.067,40.947,157.783
C06839=1040.277,229.404,-105.691,171.064,40.946,157.783
C06840=1040.270,229.156,-105.662,171.062,40.943,157.782
C06841=1040.263,228.908,-105.634,171.059,40.942,157.782
C06842=1040.257,228.659,-105.607,171.057,40.940,157.781
C06843=1040.250,228.411,-105.579,171.054,40.939,157.781
C06844=1040.243,228.163,-105.551,171.052,40.937,157.780
C06845=1040.237,227.914,-105.524,171.049,40.935,157.780
C06846=1040.230,227.666,-105.496,171.047,40.934,157.779
C06847=1040.224,227.417,-105.469,171.044,40.932,157.779
C06848=1040.217,227.168,-105.441,171.042,40.931,157.778
C06849=1040.210,226.920,-105.413,171.039,40.929,157.778
C06850=1040.204,226.672,-105.386,171.037,40.927,157.777
C06851=1040.197,226.424,-105.359,171.034,40.926,157.777
C06852=1040.190,226.175,-105.331,171.031,40.924,157.777
C06853=1040.183,225.927,-105.303,171.029,40.922,157.776
C06854=1040.177,225.679,-105.276,171.026,40.921,157.776
C06855=1040.170,225.430,-105.248,171.024,40.919,157.775
C06856=1040.164,225.181,-105.221,171.021,40.918,157.775
C06857=1040.157,224.933,-105.193,171.019,40.916,157.774
C06858=1040.150,224.684,-105.166,171.016,40.914,157.774
C06859=1040.143,224.437,-105.139,171.015,40.912,157.773
C06860=1040.137,224.188,-105.111,171.012,40.910,157.773
C06861=1040.130,223.939,-105.084,171.010,40.909,157.772
C06862=1040.124,223.691,-105.056,171.007,40.907,157.772
C06863=1040.117,223.442,-105.028,171.005,40.906,157.771
C06864=1040.110,223.194,-105.001,171.002,40.904,157.771
C06865=1040.103,222.946,-104.974,171.000,40.902,157.770
C06866=1040.097,222.697,-104.947,170.997,40.901,157.770
C06867=1040.090,222.449,-104.919,170.995,40.899,157.769
C06868=1040.084,222.201,-104.891,170.992,40.897,157.769
C06869=1040.077,221.952,-104.864,170.990,40.896,157.768
C06870=1040.071,221.703,-104.837,170.988,40.894,157.768
C06871=1040.064,221.456,-104.810,170.986,40.892,157.768
C06872=1040.057,221.207,-104.782,170.983,40.890,157.767
C06873=1040.049,220.892,-104.747,170.979,40.889,157.766
C06874=1040.041,220.578,-104.713,170.977,40.886,157.766
C06875=1040.032,220.264,-104.679,170.974,40.884,157.765
C06876=1040.024,219.949,-104.644,170.970,40.882,157.765
C06877=1040.017,219.701,-104.618,170.968,40.880,157.764
C06878=1040.011,219.453,-104.590,170.965,40.879,157.764
C06879=1040.004,219.204,-104.563,170.964,40.877,157.763
C06880=1039.997,218.956,-104.536,170.961,40.875,157.763
C06881=1039.991,218.706,-104.509,170.959,40.874,157.762
C06882=1039.984,218.459,-104.482,170.956,40.872,157.762
C06883=1039.977,218.211,-104.454,170.954,40.871,157.761
C06884=1039.971,217.962,-104.427,170.951,40.869,157.761
C06885=1039.964,217.713,-104.401,170.949,40.867,157.760
C06886=1039.957,217.464,-104.373,170.946,40.866,157.760
C06887=1039.950,217.216,-104.347,170.945,40.864,157.760
C06888=1039.944,216.968,-104.319,170.942,40.862,157.759
C06889=1039.937,216.719,-104.293,170.940,40.861,157.759
C06890=1039.930,216.471,-104.265,170.937,40.859,157.758
C06891=1039.924,216.222,-104.239,170.935,40.857,157.758
C06892=1039.917,215.974,-104.211,170.932,40.856,157.757
C06893=1039.910,215.725,-104.184,170.931,40.854,157.757
C06894=1039.904,215.478,-104.158,170.928,40.852,157.756
C06895=1039.897,215.229,-104.131,170.926,40.851,157.756
C06896=1039.890,214.980,-104.104,170.923,40.849,157.755
C06897=1039.883,214.731,-104.076,170.921,40.848,157.755
C06898=1039.877,214.483,-104.050,170.918,40.846,157.754
C06899=1039.871,214.234,-104.023,170.917,40.844,157.754
C06900=1039.864,213.986,-103.996,170.914,40.843,157.754
C06901=1039.857,213.738,-103.970,170.912,40.841,157.753
C06902=1039.851,213.489,-103.943,170.909,40.839,157.753
C06903=1039.844,213.241,-103.915,170.907,40.838,157.752
C06904=1039.838,212.992,-103.889,170.905,40.836,157.752
C06905=1039.831,212.744,-103.862,170.902,40.834,157.751
C06906=1039.825,212.496,-103.835,170.900,40.832,157.751
C06907=1039.817,212.247,-103.809,170.897,40.830,157.750
C06908=1039.811,211.998,-103.782,170.895,40.829,157.750
C06909=1039.804,211.751,-103.755,170.893,40.827,157.749
C06910=1039.798,211.502,-103.728,170.891,40.825,157.749
C06911=1039.791,211.253,-103.701,170.888,40.824,157.748
C06912=1039.785,211.004,-103.675,170.886,40.822,157.748
C06913=1039.778,210.756,-103.648,170.884,40.820,157.747
C06914=1039.770,210.508,-103.621,170.882,40.819,157.747
C06915=1039.765,210.259,-103.595,170.879,40.817,157.746
C06916=1039.758,210.010,-103.568,170.877,40.815,157.746
C06917=1039.751,209.762,-103.542,170.874,40.814,157.746
C06918=1039.745,209.513,-103.515,170.873,40.812,157.745
C06919=1039.738,209.265,-103.489,170.870,40.810,157.745
C06920=1039.732,209.017,-103.461,170.868,40.809,157.744
C06921=1039.724,208.768,-103.435,170.865,40.807,157.744
C06922=1039.717,208.519,-103.408,170.864,40.805,157.743
C06923=1039.711,208.271,-103.382,170.861,40.804,157.743
C06924=1039.704,208.022,-103.355,170.859,40.802,157.742
C06925=1039.698,207.774,-103.329,170.856,40.801,157.742
C06926=1039.691,207.525,-103.303,170.855,40.799,157.741
C06927=1039.685,207.277,-103.276,170.852,40.797,157.741
C06928=1039.678,207.028,-103.250,170.850,40.796,157.741
C06929=1039.670,206.719,-103.217,170.847,40.794,157.740
C06930=1039.660,206.411,-103.184,170.845,40.792,157.739
C06931=1039.653,206.103,-103.152,170.842,40.789,157.739
C06932=1039.644,205.793,-103.119,170.840,40.788,157.738
C06933=1039.618,204.742,-103.012,170.547,40.684,157.703
C06934=1039.612,204.494,-102.987,170.545,40.683,157.702
C06935=1039.606,204.245,-102.961,170.541,40.682,157.702
C06936=1039.600,203.996,-102.937,170.538,40.681,157.702
C06937=1039.593,203.748,-102.912,170.535,40.680,157.701
C06938=1039.587,203.499,-102.887,170.532,40.679,157.701
C06939=1039.581,203.251,-102.862,170.529,40.678,157.701
C06940=1039.575,203.002,-102.836,170.526,40.677,157.700
C06941=1039.569,202.753,-102.811,170.522,40.677,157.700
C06942=1039.563,202.504,-102.786,170.520,40.675,157.700
C06943=1039.557,202.255,-102.761,170.517,40.675,157.700
C06944=1039.551,202.007,-102.736,170.513,40.674,157.699
C06945=1039.545,201.759,-102.711,170.511,40.673,157.699
C06946=1039.539,201.509,-102.686,170.508,40.672,157.699
C06947=1039.533,201.261,-102.661,170.504,40.671,157.698
C06948=1039.526,201.012,-102.636,170.501,40.670,157.698
C06949=1039.520,200.763,-102.612,170.499,40.669,157.698
C06950=1039.514,200.514,-102.586,170.495,40.669,157.697
C06951=1039.507,200.267,-102.562,170.492,40.668,157.697
C06952=1039.501,200.018,-102.537,170.489,40.667,157.697
C06953=1039.494,199.769,-102.512,170.486,40.666,157.696
C06954=1039.488,199.520,-102.488,170.483,40.666,157.696
C06955=1039.482,199.271,-102.462,170.480,40.665,157.696
C06956=1039.476,199.022,-102.438,170.478,40.664,157.695
C06957=1039.470,198.774,-102.413,170.474,40.664,157.695
C06958=1039.463,198.525,-102.389,170.471,40.663,157.695
C06959=1039.457,198.277,-102.364,170.468,40.662,157.695
C06960=1039.451,198.028,-102.340,170.466,40.662,157.694
C06961=1039.444,197.779,-102.315,170.462,40.661,157.694
C06962=1039.439,197.530,-102.290,170.459,40.660,157.694
C06963=1039.432,197.282,-102.266,170.457,40.659,157.693
C06964=1039.426,197.033,-102.241,170.453,40.658,157.693
C06965=1039.419,196.784,-102.216,170.450,40.657,157.693
C06966=1039.414,196.536,-102.192,170.448,40.657,157.693
C06967=1039.407,196.287,-102.167,170.444,40.656,157.692
C06968=1039.401,196.038,-102.143,170.441,40.655,157.692
C06969=1039.394,195.789,-102.119,170.439,40.655,157.692
C06970=1039.389,195.541,-102.094,170.436,40.654,157.691
C06971=1039.383,195.292,-102.069,170.432,40.653,157.691
C06972=1039.376,195.044,-102.044,170.430,40.653,157.691
C06973=1039.370,194.794,-102.020,170.427,40.652,157.690
C06974=1039.364,194.546,-101.996,170.423,40.651,157.690
C06975=1039.358,194.297,-101.971,170.421,40.650,157.690
C06976=1039.351,194.048,-101.947,170.418,40.649,157.690
C06977=1039.346,193.800,-101.922,170.415,40.648,157.689
C06978=1039.339,193.551,-101.898,170.412,40.648,157.689
C06979=1039.333,193.302,-101.873,170.409,40.647,157.689
C06980=1039.327,193.054,-101.849,170.406,40.647,157.688
C06981=1039.321,192.805,-101.825,170.403,40.646,157.688
C06982=1039.314,192.556,-101.800,170.400,40.645,157.688
C06983=1039.309,192.308,-101.776,170.397,40.645,157.688
C06984=1039.302,192.059,-101.752,170.395,40.644,157.687
C06985=1039.296,191.809,-101.727,170.391,40.643,157.687
C06986=1039.290,191.562,-101.703,170.389,40.642,157.687
C06987=1039.284,191.312,-101.678,170.386,40.641,157.686
C06988=1039.278,191.064,-101.655,170.383,40.641,157.686
C06989=1039.272,190.815,-101.630,170.380,40.640,157.686
C06990=1039.266,190.566,-101.605,170.377,40.640,157.686
C06991=1039.260,190.318,-101.581,170.375,40.639,157.685
C06992=1039.254,190.069,-101.556,170.372,40.638,157.685
C06993=1039.248,189.820,-101.533,170.368,40.637,157.685
C06994=1039.241,189.536,-101.505,170.365,40.636,157.684
C06995=1039.234,189.251,-101.477,170.361,40.636,157.684
C06996=1039.227,188.968,-101.449,170.358,40.635,157.684
C06997=1039.221,188.683,-101.422,170.356,40.634,157.684
C06998=1039.214,188.434,-101.398,170.353,40.633,157.683
C06999=1039.209,188.185,-101.373,170.349,40.633,157.683
C07000=1039.202,187.936,-101.349,170.347,40.632,157.683
C07001=1039.197,187.687,-101.325,170.344,40.632,157.682
C07002=1039.190,187.439,-101.300,170.342,40.631,157.682
C07003=1039.184,187.190,-101.276,170.338,40.630,157.682
C07004=1039.178,186.942,-101.252,170.336,40.629,157.682
C07005=1039.172,186.693,-101.228,170.333,40.628,157.681
C07006=1039.166,186.444,-101.204,170.330,40.628,157.681
C07007=1039.160,186.196,-101.180,170.327,40.627,157.681
C07008=1039.154,185.946,-101.155,170.324,40.627,157.681
C07009=1039.148,185.698,-101.132,170.322,40.626,157.680
C07010=1039.142,185.449,-101.107,170.318,40.625,157.680
C07011=1039.136,185.201,-101.083,170.316,40.624,157.680
C07012=1039.131,184.952,-101.059,170.313,40.624,157.680
C07013=1039.124,184.702,-101.036,170.311,40.623,157.679
C07014=1039.119,184.454,-101.012,170.307,40.623,157.679
C07015=1039.112,184.205,-100.988,170.305,40.622,157.679
C07016=1039.107,183.956,-100.963,170.302,40.621,157.678
C07017=1039.100,183.707,-100.939,170.300,40.620,157.678
C07018=1039.095,183.459,-100.915,170.296,40.620,157.678
C07019=1039.089,183.210,-100.891,170.294,40.619,157.678
C07020=1039.082,182.961,-100.869,170.291,40.619,157.677
C07021=1039.075,182.712,-100.845,170.288,40.618,157.677
C07022=1039.069,182.464,-100.821,170.286,40.618,157.677
C07023=1039.063,182.215,-100.797,170.282,40.618,157.677
C07024=1039.057,181.966,-100.774,170.280,40.617,157.676
C07025=1039.050,181.717,-100.750,170.277,40.616,157.676
C07026=1039.044,181.469,-100.726,170.275,40.616,157.676
C07027=1039.038,181.219,-100.703,170.271,40.616,157.676
C07028=1039.032,180.971,-100.679,170.268,40.615,157.676
C07029=1039.026,180.721,-100.656,170.266,40.614,157.675
C07030=1039.020,180.473,-100.632,170.263,40.614,157.675
C07031=1039.012,180.224,-100.609,170.261,40.614,157.675
C07032=1039.006,179.975,-100.586,170.257,40.613,157.675
C07033=1039.000,179.726,-100.562,170.255,40.613,157.675
C07034=1038.994,179.478,-100.538,170.252,40.613,157.674
C07035=1038.988,179.229,-100.515,170.250,40.611,157.674
C07036=1038.981,178.980,-100.491,170.247,40.611,157.674
C07037=1038.976,178.731,-100.468,170.244,40.611,157.674
C07038=1038.969,178.482,-100.444,170.241,40.610,157.673
C07039=1038.963,178.233,-100.421,170.238,40.610,157.673
C07040=1038.956,177.985,-100.398,170.236,40.609,157.673
C07041=1038.950,177.736,-100.375,170.232,40.609,157.673
C07042=1038.944,177.488,-100.351,170.230,40.608,157.672
C07043=1038.938,177.238,-100.328,170.227,40.608,157.672
C07044=1038.932,176.990,-100.304,170.225,40.608,157.672
C07045=1038.925,176.740,-100.281,170.222,40.607,157.672
C07046=1038.919,176.492,-100.257,170.220,40.607,157.672
C07047=1038.914,176.243,-100.234,170.216,40.606,157.671
C07048=1038.906,175.994,-100.211,170.214,40.606,157.671
C07049=1038.901,175.745,-100.188,170.211,40.605,157.671
C07050=1038.895,175.497,-100.164,170.209,40.605,157.671
C07051=1038.888,175.248,-100.141,170.205,40.605,157.671
C07052=1038.883,174.999,-100.118,170.203,40.604,157.670
C07053=1038.876,174.750,-100.095,170.200,40.604,157.670
C07054=1038.870,174.501,-100.071,170.198,40.603,157.670
C07055=1038.864,174.253,-100.048,170.195,40.603,157.670
C07056=1038.858,174.004,-100.025,170.192,40.602,157.669
C07057=1038.851,173.754,-100.002,170.190,40.602,157.669
C07058=1038.845,173.470,-99.975,170.187,40.601,157.669
C07059=1038.837,173.185,-99.949,170.184,40.600,157.669
C07060=1038.831,172.901,-99.922,170.181,40.600,157.669
C07061=1038.823,172.616,-99.896,170.177,40.600,157.668
C07062=1038.817,172.367,-99.872,170.175,40.599,157.668
C07063=1038.811,172.118,-99.849,170.172,40.599,157.668
C07064=1038.805,171.869,-99.826,170.170,40.598,157.668
C07065=1038.800,171.620,-99.803,170.167,40.598,157.667
C07066=1038.793,171.372,-99.780,170.164,40.597,157.667
C07067=1038.786,171.122,-99.757,170.162,40.597,157.667
C07068=1038.781,170.874,-99.734,170.159,40.597,157.667
C07069=1038.775,170.625,-99.711,170.157,40.596,157.667
C07070=1038.769,170.376,-99.687,170.154,40.596,157.666
C07071=1038.763,170.128,-99.664,170.151,40.596,157.666
C07072=1038.756,169.878,-99.641,170.148,40.595,157.666
C07073=1038.750,169.629,-99.618,170.146,40.594,157.666
C07074=1038.744,169.381,-99.595,170.144,40.594,157.666
C07075=1038.739,169.132,-99.572,170.141,40.593,157.665
C07076=1038.733,168.883,-99.549,170.138,40.593,157.665
C07077=1038.727,168.634,-99.526,170.135,40.593,157.665
C07078=1038.720,168.385,-99.503,170.133,40.592,157.665
C07079=1038.714,168.136,-99.480,170.131,40.592,157.665
C07080=1038.708,167.888,-99.457,170.128,40.592,157.664
C07081=1038.703,167.639,-99.434,170.125,40.591,157.664
C07082=1038.696,167.389,-99.410,170.122,40.590,157.664
C07083=1038.690,167.141,-99.388,170.120,40.590,157.664
C07084=1038.684,166.892,-99.365,170.118,40.589,157.663
C07085=1038.678,166.643,-99.342,170.115,40.589,157.663
C07086=1038.673,166.394,-99.319,170.112,40.589,157.663
C07087=1038.667,166.145,-99.296,170.110,40.588,157.663
C07088=1038.660,165.897,-99.274,170.107,40.588,157.663
C07089=1038.654,165.648,-99.250,170.105,40.588,157.662
C07090=1038.648,165.399,-99.227,170.102,40.587,157.662
C07091=1038.642,165.150,-99.204,170.099,40.587,157.662
C07092=1038.637,164.901,-99.181,170.097,40.586,157.662
C07093=1038.630,164.652,-99.159,170.094,40.586,157.662
C07094=1038.624,164.403,-99.136,170.092,40.585,157.661
C07095=1038.619,164.155,-99.113,170.090,40.585,157.661
C07096=1038.613,163.906,-99.090,170.086,40.584,157.661
C07097=1038.607,163.657,-99.067,170.084,40.584,157.661
C07098=1038.601,163.408,-99.044,170.082,40.584,157.661
C07099=1038.595,163.159,-99.022,170.079,40.583,157.660
C07100=1038.589,162.910,-98.999,170.077,40.583,157.660
C07101=1038.584,162.662,-98.976,170.075,40.582,157.660
C07102=1038.578,162.413,-98.953,170.071,40.582,157.660
C07103=1038.572,162.163,-98.931,170.069,40.581,157.659
C07104=1038.566,161.915,-98.908,170.067,40.581,157.659
C07105=1038.560,161.666,-98.885,170.064,40.580,157.659
C07106=1038.555,161.417,-98.862,170.061,40.580,157.659
C07107=1038.548,161.168,-98.840,170.059,40.579,157.659
C07108=1038.542,160.919,-98.817,170.056,40.579,157.659
C07109=1038.536,160.670,-98.794,170.054,40.579,157.658
C07110=1038.530,160.421,-98.771,170.052,40.578,157.658
C07111=1038.525,160.172,-98.748,170.049,40.578,157.658
C07112=1038.518,159.923,-98.726,170.046,40.578,157.658
C07113=1038.512,159.674,-98.704,170.044,40.577,157.658
C07114=1038.506,159.425,-98.681,170.041,40.577,157.657
C07115=1038.500,159.177,-98.658,170.039,40.576,157.657
C07116=1038.494,158.927,-98.636,170.037,40.576,157.657
C07117=1038.488,158.678,-98.614,170.034,40.576,157.657
C07118=1038.481,158.430,-98.592,170.031,40.576,157.657
C07119=1038.476,158.180,-98.569,170.029,40.576,157.657
C07120=1038.469,157.932,-98.547,170.026,40.575,157.656
C07121=1038.463,157.683,-98.525,170.024,40.575,157.656
C07122=1038.456,157.397,-98.499,170.021,40.574,157.656
C07123=1038.449,157.113,-98.474,170.019,40.574,157.656
C07124=1038.442,156.827,-98.448,170.015,40.574,157.656
C07125=1038.436,156.542,-98.422,170.012,40.573,157.655
C07126=1038.429,156.293,-98.400,170.010,40.573,157.655
C07127=1038.423,156.045,-98.378,170.008,40.573,157.655
C07128=1038.418,155.795,-98.356,170.005,40.573,157.655
C07129=1038.411,155.547,-98.333,170.003,40.573,157.655
C07130=1038.405,155.298,-98.311,170.000,40.572,157.655
C07131=1038.399,155.048,-98.289,169.997,40.572,157.654
C07132=1038.393,154.800,-98.266,169.995,40.571,157.654
C07133=1038.387,154.551,-98.245,169.993,40.571,157.654
C07134=1038.381,154.302,-98.222,169.990,40.571,157.654
C07135=1038.375,154.053,-98.200,169.988,40.571,157.654
C07136=1038.368,153.804,-98.178,169.986,40.570,157.654
C07137=1038.362,153.555,-98.156,169.982,40.570,157.653
C07138=1038.356,153.306,-98.133,169.980,40.570,157.653
C07139=1038.350,153.057,-98.112,169.978,40.570,157.653
C07140=1038.344,152.808,-98.089,169.975,40.570,157.653
C07141=1038.337,152.559,-98.068,169.973,40.569,157.653
C07142=1038.331,152.310,-98.045,169.971,40.569,157.652
C07143=1038.326,152.061,-98.023,169.969,40.569,157.652
C07144=1038.319,151.812,-98.001,169.965,40.569,157.652
C07145=1038.313,151.563,-97.979,169.963,40.568,157.652
C07146=1038.307,151.314,-97.957,169.961,40.568,157.652
C07147=1038.301,151.066,-97.935,169.958,40.568,157.652
C07148=1038.295,150.816,-97.913,169.956,40.568,157.652
C07149=1038.289,150.568,-97.891,169.954,40.567,157.651
C07150=1038.283,150.319,-97.869,169.951,40.567,157.651
C07151=1038.277,150.069,-97.848,169.948,40.567,157.651
C07152=1038.270,149.821,-97.825,169.946,40.567,157.651
C07153=1038.265,149.571,-97.803,169.944,40.566,157.651
C07154=1038.259,149.322,-97.781,169.941,40.566,157.651
C07155=1038.252,149.073,-97.759,169.939,40.566,157.650
C07156=1038.247,148.825,-97.738,169.937,40.566,157.650
C07157=1038.240,148.576,-97.716,169.935,40.565,157.650
C07158=1038.234,148.327,-97.694,169.931,40.565,157.650
C07159=1038.228,148.078,-97.672,169.929,40.565,157.650
C07160=1038.222,147.829,-97.651,169.927,40.565,157.650
C07161=1038.215,147.580,-97.628,169.924,40.565,157.650
C07162=1038.210,147.331,-97.606,169.922,40.564,157.649
C07163=1038.204,147.081,-97.584,169.920,40.564,157.649
C07164=1038.198,146.833,-97.563,169.918,40.564,157.649
C07165=1038.192,146.584,-97.541,169.914,40.564,157.649
C07166=1038.185,146.335,-97.519,169.912,40.563,157.649
C07167=1038.179,146.086,-97.497,169.910,40.563,157.649
C07168=1038.173,145.837,-97.476,169.908,40.563,157.648
C07169=1038.166,145.588,-97.455,169.905,40.563,157.648
C07170=1038.160,145.339,-97.433,169.903,40.563,157.648
C07171=1038.154,145.090,-97.412,169.901,40.563,157.648
C07172=1038.148,144.842,-97.390,169.898,40.562,157.648
C07173=1038.142,144.592,-97.368,169.896,40.562,157.648
C07174=1038.136,144.343,-97.346,169.893,40.562,157.648
C07175=1038.129,144.094,-97.325,169.891,40.562,157.648
C07176=1038.123,143.845,-97.303,169.888,40.562,157.647
C07177=1038.118,143.596,-97.282,169.886,40.562,157.647
C07178=1038.112,143.347,-97.260,169.884,40.562,157.647
C07179=1038.105,143.098,-97.238,169.882,40.561,157.647
C07180=1038.099,142.849,-97.217,169.879,40.561,157.647
C07181=1038.093,142.599,-97.195,169.877,40.561,157.647
C07182=1038.087,142.351,-97.174,169.874,40.561,157.646
C07183=1038.081,142.102,-97.153,169.872,40.560,157.646
C07184=1038.074,141.853,-97.130,169.869,40.561,157.646
C07185=1038.068,141.604,-97.109,169.867,40.560,157.646
C07186=1038.062,141.318,-97.085,169.865,40.560,157.646
C07187=1038.055,141.033,-97.060,169.862,40.560,157.646
C07188=1038.048,140.747,-97.036,169.860,40.560,157.646
C07189=1038.041,140.462,-97.011,169.856,40.559,157.645
C07190=1038.035,140.213,-96.989,169.854,40.559,157.645
C07191=1038.029,139.964,-96.967,169.852,40.559,157.645
C07192=1038.023,139.715,-96.946,169.849,40.559,157.645
